ABB RAPID module: P51.mod

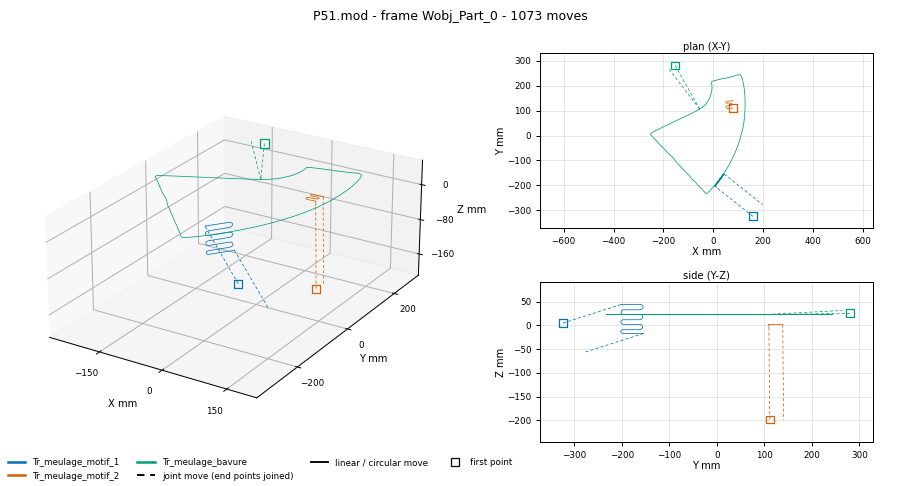
[picture p0: tool path of P51.mod in frame Wobj_Part_0, 1073 of 1081 moves have a stored position in this frame; points joined in program order, loops and branches not executed]
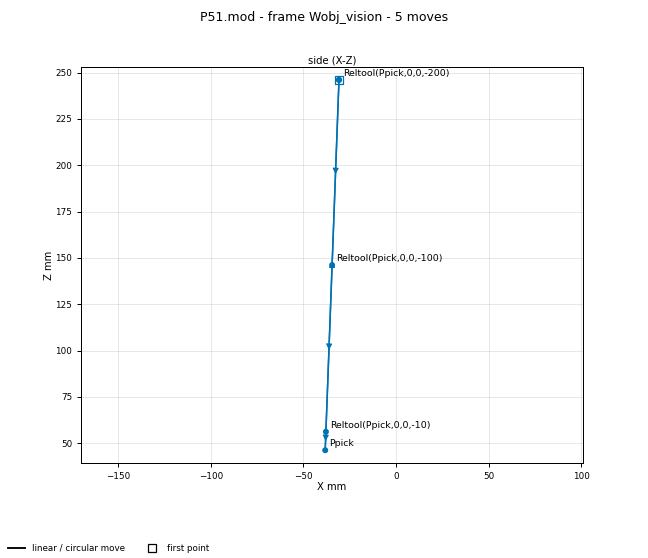
[picture p1: tool path of P51.mod in frame Wobj_vision, 5 of 1081 moves have a stored position in this frame; points joined in program order, loops and branches not executed]
MODULE P51
	LOCAL CONST Speeddata vitesse_Tronconnage :=[10, 500, 0, 0];
	LOCAL CONST Robtarget Tr_meulage_motif_1_App1 :=[[158.377655595794,-324.024414771468,4.86982949443898],[0.696320279376617,-0.571579290814731,-0.275420255163045,0.335527742350052],[0,0,0,0],[8.999999E+09,8.999999E+09,8.999999E+09,8.999999E+09,8.999999E+09,8.999999E+09]];
	LOCAL CONST Robtarget Tr_meulage_motif_1_App2 :=[[12.6243167397507,-207.899791051073,41.8973324903469],[0.696320279376617,-0.571579290814731,-0.275420255163045,0.335527742350052],[0,0,0,0],[8.999999E+09,8.999999E+09,8.999999E+09,8.999999E+09,8.999999E+09,8.999999E+09]];
	LOCAL CONST Robtarget Tr_meulage_motif_1_P0 :=[[4.95308837890625,-201.78796875,43.8461484375],[0.696320279376617,-0.571579290814731,-0.275420255163045,0.335527742350052],[0,0,0,0],[8.999999E+09,8.999999E+09,8.999999E+09,8.999999E+09,8.999999E+09,8.999999E+09]];
	LOCAL CONST Robtarget Tr_meulage_motif_1_P1 :=[[5.54933837890625,-200.985171875,43.84616796875],[0.696320279376617,-0.571579290814731,-0.275420255163045,0.335527742350052],[0,0,0,0],[8.999999E+09,8.999999E+09,8.999999E+09,8.999999E+09,8.999999E+09,8.999999E+09]];
	LOCAL CONST Robtarget Tr_meulage_motif_1_P2 :=[[6.1455888671875,-200.182375,43.8461875],[0.696320279376617,-0.571579290814731,-0.275420255163045,0.335527742350052],[0,0,0,0],[8.999999E+09,8.999999E+09,8.999999E+09,8.999999E+09,8.999999E+09,8.999999E+09]];
	LOCAL CONST Robtarget Tr_meulage_motif_1_P3 :=[[6.74183935546875,-199.379578125,43.84620703125],[0.696320279376617,-0.571579290814731,-0.275420255163045,0.335527742350052],[0,0,0,0],[8.999999E+09,8.999999E+09,8.999999E+09,8.999999E+09,8.999999E+09,8.999999E+09]];
	LOCAL CONST Robtarget Tr_meulage_motif_1_P4 :=[[7.33808935546875,-198.57678125,43.84623046875],[0.696320279376617,-0.571579290814731,-0.275420255163045,0.335527742350052],[0,0,0,0],[8.999999E+09,8.999999E+09,8.999999E+09,8.999999E+09,8.999999E+09,8.999999E+09]];
	LOCAL CONST Robtarget Tr_meulage_motif_1_P5 :=[[7.93433984375,-197.773984375,43.84625],[0.696320279376617,-0.571579290814731,-0.275420255163045,0.335527742350052],[0,0,0,0],[8.999999E+09,8.999999E+09,8.999999E+09,8.999999E+09,8.999999E+09,8.999999E+09]];
	LOCAL CONST Robtarget Tr_meulage_motif_1_P6 :=[[8.53058984375,-196.9711875,43.84626953125],[0.696320279376617,-0.571579290814731,-0.275420255163045,0.335527742350052],[0,0,0,0],[8.999999E+09,8.999999E+09,8.999999E+09,8.999999E+09,8.999999E+09,8.999999E+09]];
	LOCAL CONST Robtarget Tr_meulage_motif_1_P7 :=[[9.12683984375,-196.168390625,43.8462890625],[0.696320279376617,-0.571579290814731,-0.275420255163045,0.335527742350052],[0,0,0,0],[8.999999E+09,8.999999E+09,8.999999E+09,8.999999E+09,8.999999E+09,8.999999E+09]];
	LOCAL CONST Robtarget Tr_meulage_motif_1_P8 :=[[9.7230908203125,-195.36559375,43.84630859375],[0.696320279376617,-0.571579290814731,-0.275420255163045,0.335527742350052],[0,0,0,0],[8.999999E+09,8.999999E+09,8.999999E+09,8.999999E+09,8.999999E+09,8.999999E+09]];
	LOCAL CONST Robtarget Tr_meulage_motif_1_P9 :=[[10.3193408203125,-194.56278125,43.846328125],[0.696320279376617,-0.571579290814731,-0.275420255163045,0.335527742350052],[0,0,0,0],[8.999999E+09,8.999999E+09,8.999999E+09,8.999999E+09,8.999999E+09,8.999999E+09]];
	LOCAL CONST Robtarget Tr_meulage_motif_1_P10 :=[[10.9155908203125,-193.759984375,43.8463515625],[0.696320279376617,-0.571579290814731,-0.275420255163045,0.335527742350052],[0,0,0,0],[8.999999E+09,8.999999E+09,8.999999E+09,8.999999E+09,8.999999E+09,8.999999E+09]];
	LOCAL CONST Robtarget Tr_meulage_motif_1_P11 :=[[11.511841796875,-192.9571875,43.84637109375],[0.696320279376617,-0.571579290814731,-0.275420255163045,0.335527742350052],[0,0,0,0],[8.999999E+09,8.999999E+09,8.999999E+09,8.999999E+09,8.999999E+09,8.999999E+09]];
	LOCAL CONST Robtarget Tr_meulage_motif_1_P12 :=[[12.108091796875,-192.154390625,43.846390625],[0.696320279376617,-0.571579290814731,-0.275420255163045,0.335527742350052],[0,0,0,0],[8.999999E+09,8.999999E+09,8.999999E+09,8.999999E+09,8.999999E+09,8.999999E+09]];
	LOCAL CONST Robtarget Tr_meulage_motif_1_P13 :=[[12.704341796875,-191.35159375,43.84641015625],[0.696320279376617,-0.571579290814731,-0.275420255163045,0.335527742350052],[0,0,0,0],[8.999999E+09,8.999999E+09,8.999999E+09,8.999999E+09,8.999999E+09,8.999999E+09]];
	LOCAL CONST Robtarget Tr_meulage_motif_1_P14 :=[[13.3005927734375,-190.548796875,43.8464296875],[0.696320279376617,-0.571579290814731,-0.275420255163045,0.335527742350052],[0,0,0,0],[8.999999E+09,8.999999E+09,8.999999E+09,8.999999E+09,8.999999E+09,8.999999E+09]];
	LOCAL CONST Robtarget Tr_meulage_motif_1_P15 :=[[13.8968427734375,-189.746,43.846453125],[0.696320279376617,-0.571579290814731,-0.275420255163045,0.335527742350052],[0,0,0,0],[8.999999E+09,8.999999E+09,8.999999E+09,8.999999E+09,8.999999E+09,8.999999E+09]];
	LOCAL CONST Robtarget Tr_meulage_motif_1_P16 :=[[14.4930927734375,-188.943203125,43.84647265625],[0.696320279376617,-0.571579290814731,-0.275420255163045,0.335527742350052],[0,0,0,0],[8.999999E+09,8.999999E+09,8.999999E+09,8.999999E+09,8.999999E+09,8.999999E+09]];
	LOCAL CONST Robtarget Tr_meulage_motif_1_P17 :=[[15.0893427734375,-188.14040625,43.8464921875],[0.696320279376617,-0.571579290814731,-0.275420255163045,0.335527742350052],[0,0,0,0],[8.999999E+09,8.999999E+09,8.999999E+09,8.999999E+09,8.999999E+09,8.999999E+09]];
	LOCAL CONST Robtarget Tr_meulage_motif_1_P18 :=[[15.68559375,-187.33759375,43.84651171875],[0.696320279376617,-0.571579290814731,-0.275420255163045,0.335527742350052],[0,0,0,0],[8.999999E+09,8.999999E+09,8.999999E+09,8.999999E+09,8.999999E+09,8.999999E+09]];
	LOCAL CONST Robtarget Tr_meulage_motif_1_P19 :=[[16.28184375,-186.534796875,43.84653125],[0.696320279376617,-0.571579290814731,-0.275420255163045,0.335527742350052],[0,0,0,0],[8.999999E+09,8.999999E+09,8.999999E+09,8.999999E+09,8.999999E+09,8.999999E+09]];
	LOCAL CONST Robtarget Tr_meulage_motif_1_P20 :=[[16.87809375,-185.732,43.8465546875],[0.696320279376617,-0.571579290814731,-0.275420255163045,0.335527742350052],[0,0,0,0],[8.999999E+09,8.999999E+09,8.999999E+09,8.999999E+09,8.999999E+09,8.999999E+09]];
	LOCAL CONST Robtarget Tr_meulage_motif_1_P21 :=[[17.47434375,-184.929203125,43.84657421875],[0.696320279376617,-0.571579290814731,-0.275420255163045,0.335527742350052],[0,0,0,0],[8.999999E+09,8.999999E+09,8.999999E+09,8.999999E+09,8.999999E+09,8.999999E+09]];
	LOCAL CONST Robtarget Tr_meulage_motif_1_P22 :=[[18.07059375,-184.12640625,43.84659375],[0.696320279376617,-0.571579290814731,-0.275420255163045,0.335527742350052],[0,0,0,0],[8.999999E+09,8.999999E+09,8.999999E+09,8.999999E+09,8.999999E+09,8.999999E+09]];
	LOCAL CONST Robtarget Tr_meulage_motif_1_P23 :=[[18.666845703125,-183.323609375,43.84661328125],[0.696320279376617,-0.571579290814731,-0.275420255163045,0.335527742350052],[0,0,0,0],[8.999999E+09,8.999999E+09,8.999999E+09,8.999999E+09,8.999999E+09,8.999999E+09]];
	LOCAL CONST Robtarget Tr_meulage_motif_1_P24 :=[[19.263095703125,-182.5208125,43.8466328125],[0.696320279376617,-0.571579290814731,-0.275420255163045,0.335527742350052],[0,0,0,0],[8.999999E+09,8.999999E+09,8.999999E+09,8.999999E+09,8.999999E+09,8.999999E+09]];
	LOCAL CONST Robtarget Tr_meulage_motif_1_P25 :=[[19.859345703125,-181.718015625,43.84665234375],[0.696320279376617,-0.571579290814731,-0.275420255163045,0.335527742350052],[0,0,0,0],[8.999999E+09,8.999999E+09,8.999999E+09,8.999999E+09,8.999999E+09,8.999999E+09]];
	LOCAL CONST Robtarget Tr_meulage_motif_1_P26 :=[[20.455595703125,-180.91521875,43.84667578125],[0.696320279376617,-0.571579290814731,-0.275420255163045,0.335527742350052],[0,0,0,0],[8.999999E+09,8.999999E+09,8.999999E+09,8.999999E+09,8.999999E+09,8.999999E+09]];
	LOCAL CONST Robtarget Tr_meulage_motif_1_P27 :=[[21.051845703125,-180.11240625,43.8466953125],[0.696320279376617,-0.571579290814731,-0.275420255163045,0.335527742350052],[0,0,0,0],[8.999999E+09,8.999999E+09,8.999999E+09,8.999999E+09,8.999999E+09,8.999999E+09]];
	LOCAL CONST Robtarget Tr_meulage_motif_1_P28 :=[[21.648095703125,-179.309609375,43.84671484375],[0.696320279376617,-0.571579290814731,-0.275420255163045,0.335527742350052],[0,0,0,0],[8.999999E+09,8.999999E+09,8.999999E+09,8.999999E+09,8.999999E+09,8.999999E+09]];
	LOCAL CONST Robtarget Tr_meulage_motif_1_P29 :=[[22.24434765625,-178.5068125,43.846734375],[0.696320279376617,-0.571579290814731,-0.275420255163045,0.335527742350052],[0,0,0,0],[8.999999E+09,8.999999E+09,8.999999E+09,8.999999E+09,8.999999E+09,8.999999E+09]];
	LOCAL CONST Robtarget Tr_meulage_motif_1_P30 :=[[22.84059765625,-177.704015625,43.84675390625],[0.696320279376617,-0.571579290814731,-0.275420255163045,0.335527742350052],[0,0,0,0],[8.999999E+09,8.999999E+09,8.999999E+09,8.999999E+09,8.999999E+09,8.999999E+09]];
	LOCAL CONST Robtarget Tr_meulage_motif_1_P31 :=[[23.43684765625,-176.90121875,43.84677734375],[0.696320279376617,-0.571579290814731,-0.275420255163045,0.335527742350052],[0,0,0,0],[8.999999E+09,8.999999E+09,8.999999E+09,8.999999E+09,8.999999E+09,8.999999E+09]];
	LOCAL CONST Robtarget Tr_meulage_motif_1_P32 :=[[24.03309765625,-176.098421875,43.846796875],[0.696320279376617,-0.571579290814731,-0.275420255163045,0.335527742350052],[0,0,0,0],[8.999999E+09,8.999999E+09,8.999999E+09,8.999999E+09,8.999999E+09,8.999999E+09]];
	LOCAL CONST Robtarget Tr_meulage_motif_1_P33 :=[[24.62934765625,-175.295625,43.84681640625],[0.696320279376617,-0.571579290814731,-0.275420255163045,0.335527742350052],[0,0,0,0],[8.999999E+09,8.999999E+09,8.999999E+09,8.999999E+09,8.999999E+09,8.999999E+09]];
	LOCAL CONST Robtarget Tr_meulage_motif_1_P34 :=[[25.22559765625,-174.492828125,43.8468359375],[0.696320279376617,-0.571579290814731,-0.275420255163045,0.335527742350052],[0,0,0,0],[8.999999E+09,8.999999E+09,8.999999E+09,8.999999E+09,8.999999E+09,8.999999E+09]];
	LOCAL CONST Robtarget Tr_meulage_motif_1_P35 :=[[25.82184765625,-173.69003125,43.84685546875],[0.696320279376617,-0.571579290814731,-0.275420255163045,0.335527742350052],[0,0,0,0],[8.999999E+09,8.999999E+09,8.999999E+09,8.999999E+09,8.999999E+09,8.999999E+09]];
	LOCAL CONST Robtarget Tr_meulage_motif_1_P36 :=[[26.418099609375,-172.887234375,43.84687890625],[0.696320279376617,-0.571579290814731,-0.275420255163045,0.335527742350052],[0,0,0,0],[8.999999E+09,8.999999E+09,8.999999E+09,8.999999E+09,8.999999E+09,8.999999E+09]];
	LOCAL CONST Robtarget Tr_meulage_motif_1_P37 :=[[27.014349609375,-172.084421875,43.8468984375],[0.696320279376617,-0.571579290814731,-0.275420255163045,0.335527742350052],[0,0,0,0],[8.999999E+09,8.999999E+09,8.999999E+09,8.999999E+09,8.999999E+09,8.999999E+09]];
	LOCAL CONST Robtarget Tr_meulage_motif_1_P38 :=[[27.610599609375,-171.281625,43.84691796875],[0.696320279376617,-0.571579290814731,-0.275420255163045,0.335527742350052],[0,0,0,0],[8.999999E+09,8.999999E+09,8.999999E+09,8.999999E+09,8.999999E+09,8.999999E+09]];
	LOCAL CONST Robtarget Tr_meulage_motif_1_P39 :=[[28.206849609375,-170.478828125,43.8469375],[0.696320279376617,-0.571579290814731,-0.275420255163045,0.335527742350052],[0,0,0,0],[8.999999E+09,8.999999E+09,8.999999E+09,8.999999E+09,8.999999E+09,8.999999E+09]];
	LOCAL CONST Robtarget Tr_meulage_motif_1_P40 :=[[28.803099609375,-169.67603125,43.84695703125],[0.696320279376617,-0.571579290814731,-0.275420255163045,0.335527742350052],[0,0,0,0],[8.999999E+09,8.999999E+09,8.999999E+09,8.999999E+09,8.999999E+09,8.999999E+09]];
	LOCAL CONST Robtarget Tr_meulage_motif_1_P41 :=[[29.399349609375,-168.873234375,43.8469765625],[0.696320279376617,-0.571579290814731,-0.275420255163045,0.335527742350052],[0,0,0,0],[8.999999E+09,8.999999E+09,8.999999E+09,8.999999E+09,8.999999E+09,8.999999E+09]];
	LOCAL CONST Robtarget Tr_meulage_motif_1_P42 :=[[29.995599609375,-168.0704375,43.847],[0.696320279376617,-0.571579290814731,-0.275420255163045,0.335527742350052],[0,0,0,0],[8.999999E+09,8.999999E+09,8.999999E+09,8.999999E+09,8.999999E+09,8.999999E+09]];
	LOCAL CONST Robtarget Tr_meulage_motif_1_P43 :=[[30.5918515625,-167.267640625,43.84701953125],[0.696320279376617,-0.571579290814731,-0.275420255163045,0.335527742350052],[0,0,0,0],[8.999999E+09,8.999999E+09,8.999999E+09,8.999999E+09,8.999999E+09,8.999999E+09]];
	LOCAL CONST Robtarget Tr_meulage_motif_1_P44 :=[[31.1881015625,-166.46484375,43.8470390625],[0.696320279376617,-0.571579290814731,-0.275420255163045,0.335527742350052],[0,0,0,0],[8.999999E+09,8.999999E+09,8.999999E+09,8.999999E+09,8.999999E+09,8.999999E+09]];
	LOCAL CONST Robtarget Tr_meulage_motif_1_P45 :=[[31.7843515625,-165.662046875,43.84705859375],[0.696320279376617,-0.571579290814731,-0.275420255163045,0.335527742350052],[0,0,0,0],[8.999999E+09,8.999999E+09,8.999999E+09,8.999999E+09,8.999999E+09,8.999999E+09]];
	LOCAL CONST Robtarget Tr_meulage_motif_1_P46 :=[[32.3806015625,-164.859234375,43.847078125],[0.696320279376617,-0.571579290814731,-0.275420255163045,0.335527742350052],[0,0,0,0],[8.999999E+09,8.999999E+09,8.999999E+09,8.999999E+09,8.999999E+09,8.999999E+09]];
	LOCAL CONST Robtarget Tr_meulage_motif_1_P47 :=[[32.9768515625,-164.0564375,43.8471015625],[0.696320279376617,-0.571579290814731,-0.275420255163045,0.335527742350052],[0,0,0,0],[8.999999E+09,8.999999E+09,8.999999E+09,8.999999E+09,8.999999E+09,8.999999E+09]];
	LOCAL CONST Robtarget Tr_meulage_motif_1_P48 :=[[33.5731015625,-163.253640625,43.84712109375],[0.696320279376617,-0.571579290814731,-0.275420255163045,0.335527742350052],[0,0,0,0],[8.999999E+09,8.999999E+09,8.999999E+09,8.999999E+09,8.999999E+09,8.999999E+09]];
	LOCAL CONST Robtarget Tr_meulage_motif_1_P49 :=[[34.1693515625,-162.45084375,43.847140625],[0.696320279376617,-0.571579290814731,-0.275420255163045,0.335527742350052],[0,0,0,0],[8.999999E+09,8.999999E+09,8.999999E+09,8.999999E+09,8.999999E+09,8.999999E+09]];
	LOCAL CONST Robtarget Tr_meulage_motif_1_P50 :=[[34.7656015625,-161.648046875,43.84716015625],[0.696320279376617,-0.571579290814731,-0.275420255163045,0.335527742350052],[0,0,0,0],[8.999999E+09,8.999999E+09,8.999999E+09,8.999999E+09,8.999999E+09,8.999999E+09]];
	LOCAL CONST Robtarget Tr_meulage_motif_1_P51 :=[[35.3618515625,-160.84525,43.8471796875],[0.696320279376617,-0.571579290814731,-0.275420255163045,0.335527742350052],[0,0,0,0],[8.999999E+09,8.999999E+09,8.999999E+09,8.999999E+09,8.999999E+09,8.999999E+09]];
	LOCAL CONST Robtarget Tr_meulage_motif_1_P52 :=[[35.957796875,-160.051484375,43.7367265625],[0.696320279376617,-0.571579290814731,-0.275420255163045,0.335527742350052],[0,0,0,0],[8.999999E+09,8.999999E+09,8.999999E+09,8.999999E+09,8.999999E+09,8.999999E+09]];
	LOCAL CONST Robtarget Tr_meulage_motif_1_P53 :=[[36.53003125,-159.297484375,43.52578515625],[0.696320279376617,-0.571579290814731,-0.275420255163045,0.335527742350052],[0,0,0,0],[8.999999E+09,8.999999E+09,8.999999E+09,8.999999E+09,8.999999E+09,8.999999E+09]];
	LOCAL CONST Robtarget Tr_meulage_motif_1_P54 :=[[37.04861328125,-158.620453125,43.25425390625],[0.696320279376617,-0.571579290814731,-0.275420255163045,0.335527742350052],[0,0,0,0],[8.999999E+09,8.999999E+09,8.999999E+09,8.999999E+09,8.999999E+09,8.999999E+09]];
	LOCAL CONST Robtarget Tr_meulage_motif_1_P55 :=[[37.5060625,-158.026046875,42.97862890625],[0.696320279376617,-0.571579290814731,-0.275420255163045,0.335527742350052],[0,0,0,0],[8.999999E+09,8.999999E+09,8.999999E+09,8.999999E+09,8.999999E+09,8.999999E+09]];
	LOCAL CONST Robtarget Tr_meulage_motif_1_P56 :=[[38.1855703125,-157.1591875,42.36319140625],[0.696320279376617,-0.571579290814731,-0.275420255163045,0.335527742350052],[0,0,0,0],[8.999999E+09,8.999999E+09,8.999999E+09,8.999999E+09,8.999999E+09,8.999999E+09]];
	LOCAL CONST Robtarget Tr_meulage_motif_1_P57 :=[[38.8276953125,-156.3606875,41.51647265625],[0.696320279376617,-0.571579290814731,-0.275420255163045,0.335527742350052],[0,0,0,0],[8.999999E+09,8.999999E+09,8.999999E+09,8.999999E+09,8.999999E+09,8.999999E+09]];
	LOCAL CONST Robtarget Tr_meulage_motif_1_P58 :=[[39.371328125,-155.7085625,40.49372265625],[0.696320279376617,-0.571579290814731,-0.275420255163045,0.335527742350052],[0,0,0,0],[8.999999E+09,8.999999E+09,8.999999E+09,8.999999E+09,8.999999E+09,8.999999E+09]];
	LOCAL CONST Robtarget Tr_meulage_motif_1_P59 :=[[39.7040546875,-155.347578125,39.37875],[0.696320279376617,-0.571579290814731,-0.275420255163045,0.335527742350052],[0,0,0,0],[8.999999E+09,8.999999E+09,8.999999E+09,8.999999E+09,8.999999E+09,8.999999E+09]];
	LOCAL CONST Robtarget Tr_meulage_motif_1_P60 :=[[39.74616796875,-155.345125,38.68353515625],[0.696320279376617,-0.571579290814731,-0.275420255163045,0.335527742350052],[0,0,0,0],[8.999999E+09,8.999999E+09,8.999999E+09,8.999999E+09,8.999999E+09,8.999999E+09]];
	LOCAL CONST Robtarget Tr_meulage_motif_1_P61 :=[[39.7708515625,-155.363453125,38.023],[0.696320279376617,-0.571579290814731,-0.275420255163045,0.335527742350052],[0,0,0,0],[8.999999E+09,8.999999E+09,8.999999E+09,8.999999E+09,8.999999E+09,8.999999E+09]];
	LOCAL CONST Robtarget Tr_meulage_motif_1_P62 :=[[39.76280859375,-155.4258125,37.36262109375],[0.696320279376617,-0.571579290814731,-0.275420255163045,0.335527742350052],[0,0,0,0],[8.999999E+09,8.999999E+09,8.999999E+09,8.999999E+09,8.999999E+09,8.999999E+09]];
	LOCAL CONST Robtarget Tr_meulage_motif_1_P63 :=[[39.50687109375,-155.856296875,36.26205078125],[0.696320279376617,-0.571579290814731,-0.275420255163045,0.335527742350052],[0,0,0,0],[8.999999E+09,8.999999E+09,8.999999E+09,8.999999E+09,8.999999E+09,8.999999E+09]];
	LOCAL CONST Robtarget Tr_meulage_motif_1_P64 :=[[39.03368359375,-156.571875,35.25649609375],[0.696320279376617,-0.571579290814731,-0.275420255163045,0.335527742350052],[0,0,0,0],[8.999999E+09,8.999999E+09,8.999999E+09,8.999999E+09,8.999999E+09,8.999999E+09]];
	LOCAL CONST Robtarget Tr_meulage_motif_1_P65 :=[[38.4544140625,-157.416421875,34.42849609375],[0.696320279376617,-0.571579290814731,-0.275420255163045,0.335527742350052],[0,0,0,0],[8.999999E+09,8.999999E+09,8.999999E+09,8.999999E+09,8.999999E+09,8.999999E+09]];
	LOCAL CONST Robtarget Tr_meulage_motif_1_P66 :=[[38.0595078125,-157.978984375,34.03316015625],[0.696320279376617,-0.571579290814731,-0.275420255163045,0.335527742350052],[0,0,0,0],[8.999999E+09,8.999999E+09,8.999999E+09,8.999999E+09,8.999999E+09,8.999999E+09]];
	LOCAL CONST Robtarget Tr_meulage_motif_1_P67 :=[[37.38715234375,-158.92225,33.5461328125],[0.696320279376617,-0.571579290814731,-0.275420255163045,0.335527742350052],[0,0,0,0],[8.999999E+09,8.999999E+09,8.999999E+09,8.999999E+09,8.999999E+09,8.999999E+09]];
	LOCAL CONST Robtarget Tr_meulage_motif_1_P68 :=[[36.89316015625,-159.607953125,33.28230859375],[0.696320279376617,-0.571579290814731,-0.275420255163045,0.335527742350052],[0,0,0,0],[8.999999E+09,8.999999E+09,8.999999E+09,8.999999E+09,8.999999E+09,8.999999E+09]];
	LOCAL CONST Robtarget Tr_meulage_motif_1_P69 :=[[36.34508984375,-160.361828125,33.0780390625],[0.696320279376617,-0.571579290814731,-0.275420255163045,0.335527742350052],[0,0,0,0],[8.999999E+09,8.999999E+09,8.999999E+09,8.999999E+09,8.999999E+09,8.999999E+09]];
	LOCAL CONST Robtarget Tr_meulage_motif_1_P70 :=[[35.76388671875,-161.152828125,32.96954296875],[0.696320279376617,-0.571579290814731,-0.275420255163045,0.335527742350052],[0,0,0,0],[8.999999E+09,8.999999E+09,8.999999E+09,8.999999E+09,8.999999E+09,8.999999E+09]];
	LOCAL CONST Robtarget Tr_meulage_motif_1_P71 :=[[35.17619921875,-161.95271875,32.85905078125],[0.696320279376617,-0.571579290814731,-0.275420255163045,0.335527742350052],[0,0,0,0],[8.999999E+09,8.999999E+09,8.999999E+09,8.999999E+09,8.999999E+09,8.999999E+09]];
	LOCAL CONST Robtarget Tr_meulage_motif_1_P72 :=[[34.57994921875,-162.755515625,32.85903125],[0.696320279376617,-0.571579290814731,-0.275420255163045,0.335527742350052],[0,0,0,0],[8.999999E+09,8.999999E+09,8.999999E+09,8.999999E+09,8.999999E+09,8.999999E+09]];
	LOCAL CONST Robtarget Tr_meulage_motif_1_P73 :=[[33.9836953125,-163.558328125,32.8590078125],[0.696320279376617,-0.571579290814731,-0.275420255163045,0.335527742350052],[0,0,0,0],[8.999999E+09,8.999999E+09,8.999999E+09,8.999999E+09,8.999999E+09,8.999999E+09]];
	LOCAL CONST Robtarget Tr_meulage_motif_1_P74 :=[[33.3874453125,-164.361125,32.85898828125],[0.696320279376617,-0.571579290814731,-0.275420255163045,0.335527742350052],[0,0,0,0],[8.999999E+09,8.999999E+09,8.999999E+09,8.999999E+09,8.999999E+09,8.999999E+09]];
	LOCAL CONST Robtarget Tr_meulage_motif_1_P75 :=[[32.7911953125,-165.163921875,32.85896875],[0.696320279376617,-0.571579290814731,-0.275420255163045,0.335527742350052],[0,0,0,0],[8.999999E+09,8.999999E+09,8.999999E+09,8.999999E+09,8.999999E+09,8.999999E+09]];
	LOCAL CONST Robtarget Tr_meulage_motif_1_P76 :=[[32.1949453125,-165.96671875,32.85894921875],[0.696320279376617,-0.571579290814731,-0.275420255163045,0.335527742350052],[0,0,0,0],[8.999999E+09,8.999999E+09,8.999999E+09,8.999999E+09,8.999999E+09,8.999999E+09]];
	LOCAL CONST Robtarget Tr_meulage_motif_1_P77 :=[[31.5986953125,-166.769515625,32.8589296875],[0.696320279376617,-0.571579290814731,-0.275420255163045,0.335527742350052],[0,0,0,0],[8.999999E+09,8.999999E+09,8.999999E+09,8.999999E+09,8.999999E+09,8.999999E+09]];
	LOCAL CONST Robtarget Tr_meulage_motif_1_P78 :=[[31.0024453125,-167.5723125,32.85890625],[0.696320279376617,-0.571579290814731,-0.275420255163045,0.335527742350052],[0,0,0,0],[8.999999E+09,8.999999E+09,8.999999E+09,8.999999E+09,8.999999E+09,8.999999E+09]];
	LOCAL CONST Robtarget Tr_meulage_motif_1_P79 :=[[30.4061953125,-168.375109375,32.85888671875],[0.696320279376617,-0.571579290814731,-0.275420255163045,0.335527742350052],[0,0,0,0],[8.999999E+09,8.999999E+09,8.999999E+09,8.999999E+09,8.999999E+09,8.999999E+09]];
	LOCAL CONST Robtarget Tr_meulage_motif_1_P80 :=[[29.8099453125,-169.17790625,32.8588671875],[0.696320279376617,-0.571579290814731,-0.275420255163045,0.335527742350052],[0,0,0,0],[8.999999E+09,8.999999E+09,8.999999E+09,8.999999E+09,8.999999E+09,8.999999E+09]];
	LOCAL CONST Robtarget Tr_meulage_motif_1_P81 :=[[29.2136953125,-169.980703125,32.85884765625],[0.696320279376617,-0.571579290814731,-0.275420255163045,0.335527742350052],[0,0,0,0],[8.999999E+09,8.999999E+09,8.999999E+09,8.999999E+09,8.999999E+09,8.999999E+09]];
	LOCAL CONST Robtarget Tr_meulage_motif_1_P82 :=[[28.6174453125,-170.783515625,32.858828125],[0.696320279376617,-0.571579290814731,-0.275420255163045,0.335527742350052],[0,0,0,0],[8.999999E+09,8.999999E+09,8.999999E+09,8.999999E+09,8.999999E+09,8.999999E+09]];
	LOCAL CONST Robtarget Tr_meulage_motif_1_P83 :=[[28.021193359375,-171.5863125,32.8588046875],[0.696320279376617,-0.571579290814731,-0.275420255163045,0.335527742350052],[0,0,0,0],[8.999999E+09,8.999999E+09,8.999999E+09,8.999999E+09,8.999999E+09,8.999999E+09]];
	LOCAL CONST Robtarget Tr_meulage_motif_1_P84 :=[[27.424943359375,-172.389109375,32.85878515625],[0.696320279376617,-0.571579290814731,-0.275420255163045,0.335527742350052],[0,0,0,0],[8.999999E+09,8.999999E+09,8.999999E+09,8.999999E+09,8.999999E+09,8.999999E+09]];
	LOCAL CONST Robtarget Tr_meulage_motif_1_P85 :=[[26.828693359375,-173.19190625,32.858765625],[0.696320279376617,-0.571579290814731,-0.275420255163045,0.335527742350052],[0,0,0,0],[8.999999E+09,8.999999E+09,8.999999E+09,8.999999E+09,8.999999E+09,8.999999E+09]];
	LOCAL CONST Robtarget Tr_meulage_motif_1_P86 :=[[26.232443359375,-173.994703125,32.85874609375],[0.696320279376617,-0.571579290814731,-0.275420255163045,0.335527742350052],[0,0,0,0],[8.999999E+09,8.999999E+09,8.999999E+09,8.999999E+09,8.999999E+09,8.999999E+09]];
	LOCAL CONST Robtarget Tr_meulage_motif_1_P87 :=[[25.636193359375,-174.7975,32.8587265625],[0.696320279376617,-0.571579290814731,-0.275420255163045,0.335527742350052],[0,0,0,0],[8.999999E+09,8.999999E+09,8.999999E+09,8.999999E+09,8.999999E+09,8.999999E+09]];
	LOCAL CONST Robtarget Tr_meulage_motif_1_P88 :=[[25.039943359375,-175.600296875,32.85870703125],[0.696320279376617,-0.571579290814731,-0.275420255163045,0.335527742350052],[0,0,0,0],[8.999999E+09,8.999999E+09,8.999999E+09,8.999999E+09,8.999999E+09,8.999999E+09]];
	LOCAL CONST Robtarget Tr_meulage_motif_1_P89 :=[[24.44369140625,-176.40309375,32.85868359375],[0.696320279376617,-0.571579290814731,-0.275420255163045,0.335527742350052],[0,0,0,0],[8.999999E+09,8.999999E+09,8.999999E+09,8.999999E+09,8.999999E+09,8.999999E+09]];
	LOCAL CONST Robtarget Tr_meulage_motif_1_P90 :=[[23.84744140625,-177.205890625,32.8586640625],[0.696320279376617,-0.571579290814731,-0.275420255163045,0.335527742350052],[0,0,0,0],[8.999999E+09,8.999999E+09,8.999999E+09,8.999999E+09,8.999999E+09,8.999999E+09]];
	LOCAL CONST Robtarget Tr_meulage_motif_1_P91 :=[[23.25119140625,-178.008703125,32.85864453125],[0.696320279376617,-0.571579290814731,-0.275420255163045,0.335527742350052],[0,0,0,0],[8.999999E+09,8.999999E+09,8.999999E+09,8.999999E+09,8.999999E+09,8.999999E+09]];
	LOCAL CONST Robtarget Tr_meulage_motif_1_P92 :=[[22.65494140625,-178.8115,32.858625],[0.696320279376617,-0.571579290814731,-0.275420255163045,0.335527742350052],[0,0,0,0],[8.999999E+09,8.999999E+09,8.999999E+09,8.999999E+09,8.999999E+09,8.999999E+09]];
	LOCAL CONST Robtarget Tr_meulage_motif_1_P93 :=[[22.05869140625,-179.614296875,32.85860546875],[0.696320279376617,-0.571579290814731,-0.275420255163045,0.335527742350052],[0,0,0,0],[8.999999E+09,8.999999E+09,8.999999E+09,8.999999E+09,8.999999E+09,8.999999E+09]];
	LOCAL CONST Robtarget Tr_meulage_motif_1_P94 :=[[21.46244140625,-180.41709375,32.85858203125],[0.696320279376617,-0.571579290814731,-0.275420255163045,0.335527742350052],[0,0,0,0],[8.999999E+09,8.999999E+09,8.999999E+09,8.999999E+09,8.999999E+09,8.999999E+09]];
	LOCAL CONST Robtarget Tr_meulage_motif_1_P95 :=[[20.86619140625,-181.219890625,32.8585625],[0.696320279376617,-0.571579290814731,-0.275420255163045,0.335527742350052],[0,0,0,0],[8.999999E+09,8.999999E+09,8.999999E+09,8.999999E+09,8.999999E+09,8.999999E+09]];
	LOCAL CONST Robtarget Tr_meulage_motif_1_P96 :=[[20.269939453125,-182.0226875,32.85854296875],[0.696320279376617,-0.571579290814731,-0.275420255163045,0.335527742350052],[0,0,0,0],[8.999999E+09,8.999999E+09,8.999999E+09,8.999999E+09,8.999999E+09,8.999999E+09]];
	LOCAL CONST Robtarget Tr_meulage_motif_1_P97 :=[[19.673689453125,-182.825484375,32.8585234375],[0.696320279376617,-0.571579290814731,-0.275420255163045,0.335527742350052],[0,0,0,0],[8.999999E+09,8.999999E+09,8.999999E+09,8.999999E+09,8.999999E+09,8.999999E+09]];
	LOCAL CONST Robtarget Tr_meulage_motif_1_P98 :=[[19.077439453125,-183.62828125,32.85850390625],[0.696320279376617,-0.571579290814731,-0.275420255163045,0.335527742350052],[0,0,0,0],[8.999999E+09,8.999999E+09,8.999999E+09,8.999999E+09,8.999999E+09,8.999999E+09]];
	LOCAL CONST Robtarget Tr_meulage_motif_1_P99 :=[[18.481189453125,-184.431078125,32.85848046875],[0.696320279376617,-0.571579290814731,-0.275420255163045,0.335527742350052],[0,0,0,0],[8.999999E+09,8.999999E+09,8.999999E+09,8.999999E+09,8.999999E+09,8.999999E+09]];
	LOCAL CONST Robtarget Tr_meulage_motif_1_P100 :=[[17.884939453125,-185.233890625,32.8584609375],[0.696320279376617,-0.571579290814731,-0.275420255163045,0.335527742350052],[0,0,0,0],[8.999999E+09,8.999999E+09,8.999999E+09,8.999999E+09,8.999999E+09,8.999999E+09]];
	LOCAL CONST Robtarget Tr_meulage_motif_1_P101 :=[[17.288689453125,-186.0366875,32.85844140625],[0.696320279376617,-0.571579290814731,-0.275420255163045,0.335527742350052],[0,0,0,0],[8.999999E+09,8.999999E+09,8.999999E+09,8.999999E+09,8.999999E+09,8.999999E+09]];
	LOCAL CONST Robtarget Tr_meulage_motif_1_P102 :=[[16.692439453125,-186.839484375,32.858421875],[0.696320279376617,-0.571579290814731,-0.275420255163045,0.335527742350052],[0,0,0,0],[8.999999E+09,8.999999E+09,8.999999E+09,8.999999E+09,8.999999E+09,8.999999E+09]];
	LOCAL CONST Robtarget Tr_meulage_motif_1_P103 :=[[16.0961884765625,-187.64228125,32.85840234375],[0.696320279376617,-0.571579290814731,-0.275420255163045,0.335527742350052],[0,0,0,0],[8.999999E+09,8.999999E+09,8.999999E+09,8.999999E+09,8.999999E+09,8.999999E+09]];
	LOCAL CONST Robtarget Tr_meulage_motif_1_P104 :=[[15.4999384765625,-188.445078125,32.8583828125],[0.696320279376617,-0.571579290814731,-0.275420255163045,0.335527742350052],[0,0,0,0],[8.999999E+09,8.999999E+09,8.999999E+09,8.999999E+09,8.999999E+09,8.999999E+09]];
	LOCAL CONST Robtarget Tr_meulage_motif_1_P105 :=[[14.9036875,-189.247875,32.858359375],[0.696320279376617,-0.571579290814731,-0.275420255163045,0.335527742350052],[0,0,0,0],[8.999999E+09,8.999999E+09,8.999999E+09,8.999999E+09,8.999999E+09,8.999999E+09]];
	LOCAL CONST Robtarget Tr_meulage_motif_1_P106 :=[[14.3074375,-190.050671875,32.85833984375],[0.696320279376617,-0.571579290814731,-0.275420255163045,0.335527742350052],[0,0,0,0],[8.999999E+09,8.999999E+09,8.999999E+09,8.999999E+09,8.999999E+09,8.999999E+09]];
	LOCAL CONST Robtarget Tr_meulage_motif_1_P107 :=[[13.7111875,-190.85346875,32.8583203125],[0.696320279376617,-0.571579290814731,-0.275420255163045,0.335527742350052],[0,0,0,0],[8.999999E+09,8.999999E+09,8.999999E+09,8.999999E+09,8.999999E+09,8.999999E+09]];
	LOCAL CONST Robtarget Tr_meulage_motif_1_P108 :=[[13.1149365234375,-191.656265625,32.85830078125],[0.696320279376617,-0.571579290814731,-0.275420255163045,0.335527742350052],[0,0,0,0],[8.999999E+09,8.999999E+09,8.999999E+09,8.999999E+09,8.999999E+09,8.999999E+09]];
	LOCAL CONST Robtarget Tr_meulage_motif_1_P109 :=[[12.5186865234375,-192.459078125,32.85828125],[0.696320279376617,-0.571579290814731,-0.275420255163045,0.335527742350052],[0,0,0,0],[8.999999E+09,8.999999E+09,8.999999E+09,8.999999E+09,8.999999E+09,8.999999E+09]];
	LOCAL CONST Robtarget Tr_meulage_motif_1_P110 :=[[11.9224365234375,-193.261875,32.8582578125],[0.696320279376617,-0.571579290814731,-0.275420255163045,0.335527742350052],[0,0,0,0],[8.999999E+09,8.999999E+09,8.999999E+09,8.999999E+09,8.999999E+09,8.999999E+09]];
	LOCAL CONST Robtarget Tr_meulage_motif_1_P111 :=[[11.326185546875,-194.064671875,32.85823828125],[0.696320279376617,-0.571579290814731,-0.275420255163045,0.335527742350052],[0,0,0,0],[8.999999E+09,8.999999E+09,8.999999E+09,8.999999E+09,8.999999E+09,8.999999E+09]];
	LOCAL CONST Robtarget Tr_meulage_motif_1_P112 :=[[10.729935546875,-194.86746875,32.85821875],[0.696320279376617,-0.571579290814731,-0.275420255163045,0.335527742350052],[0,0,0,0],[8.999999E+09,8.999999E+09,8.999999E+09,8.999999E+09,8.999999E+09,8.999999E+09]];
	LOCAL CONST Robtarget Tr_meulage_motif_1_P113 :=[[10.133685546875,-195.670265625,32.85819921875],[0.696320279376617,-0.571579290814731,-0.275420255163045,0.335527742350052],[0,0,0,0],[8.999999E+09,8.999999E+09,8.999999E+09,8.999999E+09,8.999999E+09,8.999999E+09]];
	LOCAL CONST Robtarget Tr_meulage_motif_1_P114 :=[[9.537435546875,-196.4730625,32.8581796875],[0.696320279376617,-0.571579290814731,-0.275420255163045,0.335527742350052],[0,0,0,0],[8.999999E+09,8.999999E+09,8.999999E+09,8.999999E+09,8.999999E+09,8.999999E+09]];
	LOCAL CONST Robtarget Tr_meulage_motif_1_P115 :=[[8.9497470703125,-197.272953125,32.74768359375],[0.696320279376617,-0.571579290814731,-0.275420255163045,0.335527742350052],[0,0,0,0],[8.999999E+09,8.999999E+09,8.999999E+09,8.999999E+09,8.999999E+09,8.999999E+09]];
	LOCAL CONST Robtarget Tr_meulage_motif_1_P116 :=[[8.393279296875,-198.03865625,32.536705078125],[0.696320279376617,-0.571579290814731,-0.275420255163045,0.335527742350052],[0,0,0,0],[8.999999E+09,8.999999E+09,8.999999E+09,8.999999E+09,8.999999E+09,8.999999E+09]];
	LOCAL CONST Robtarget Tr_meulage_motif_1_P117 :=[[7.89499267578125,-198.73075,32.265138671875],[0.696320279376617,-0.571579290814731,-0.275420255163045,0.335527742350052],[0,0,0,0],[8.999999E+09,8.999999E+09,8.999999E+09,8.999999E+09,8.999999E+09,8.999999E+09]];
	LOCAL CONST Robtarget Tr_meulage_motif_1_P118 :=[[7.48211376953125,-199.310359375,31.961296875],[0.696320279376617,-0.571579290814731,-0.275420255163045,0.335527742350052],[0,0,0,0],[8.999999E+09,8.999999E+09,8.999999E+09,8.999999E+09,8.999999E+09,8.999999E+09]];
	LOCAL CONST Robtarget Tr_meulage_motif_1_P119 :=[[6.8900419921875,-200.1591875,31.2994609375],[0.696320279376617,-0.571579290814731,-0.275420255163045,0.335527742350052],[0,0,0,0],[8.999999E+09,8.999999E+09,8.999999E+09,8.999999E+09,8.999999E+09,8.999999E+09]];
	LOCAL CONST Robtarget Tr_meulage_motif_1_P120 :=[[6.385927734375,-200.908234375,30.398478515625],[0.696320279376617,-0.571579290814731,-0.275420255163045,0.335527742350052],[0,0,0,0],[8.999999E+09,8.999999E+09,8.999999E+09,8.999999E+09,8.999999E+09,8.999999E+09]];
	LOCAL CONST Robtarget Tr_meulage_motif_1_P121 :=[[6.10599755859375,-201.3666875,29.353568359375],[0.696320279376617,-0.571579290814731,-0.275420255163045,0.335527742350052],[0,0,0,0],[8.999999E+09,8.999999E+09,8.999999E+09,8.999999E+09,8.999999E+09,8.999999E+09]];
	LOCAL CONST Robtarget Tr_meulage_motif_1_P122 :=[[6.021697265625,-201.53421875,28.66109375],[0.696320279376617,-0.571579290814731,-0.275420255163045,0.335527742350052],[0,0,0,0],[8.999999E+09,8.999999E+09,8.999999E+09,8.999999E+09,8.999999E+09,8.999999E+09]];
	LOCAL CONST Robtarget Tr_meulage_motif_1_P123 :=[[6.0123720703125,-201.6068125,27.89192578125],[0.696320279376617,-0.571579290814731,-0.275420255163045,0.335527742350052],[0,0,0,0],[8.999999E+09,8.999999E+09,8.999999E+09,8.999999E+09,8.999999E+09,8.999999E+09]];
	LOCAL CONST Robtarget Tr_meulage_motif_1_P124 :=[[6.0810205078125,-201.574390625,27.122884765625],[0.696320279376617,-0.571579290814731,-0.275420255163045,0.335527742350052],[0,0,0,0],[8.999999E+09,8.999999E+09,8.999999E+09,8.999999E+09,8.999999E+09,8.999999E+09]];
	LOCAL CONST Robtarget Tr_meulage_motif_1_P125 :=[[6.37257080078125,-201.268234375,26.01583984375],[0.696320279376617,-0.571579290814731,-0.275420255163045,0.335527742350052],[0,0,0,0],[8.999999E+09,8.999999E+09,8.999999E+09,8.999999E+09,8.999999E+09,8.999999E+09]];
	LOCAL CONST Robtarget Tr_meulage_motif_1_P126 :=[[6.641466796875,-200.951859375,25.430794921875],[0.696320279376617,-0.571579290814731,-0.275420255163045,0.335527742350052],[0,0,0,0],[8.999999E+09,8.999999E+09,8.999999E+09,8.999999E+09,8.999999E+09,8.999999E+09]];
	LOCAL CONST Robtarget Tr_meulage_motif_1_P127 :=[[7.20352880859375,-200.264234375,24.544646484375],[0.696320279376617,-0.571579290814731,-0.275420255163045,0.335527742350052],[0,0,0,0],[8.999999E+09,8.999999E+09,8.999999E+09,8.999999E+09,8.999999E+09,8.999999E+09]];
	LOCAL CONST Robtarget Tr_meulage_motif_1_P128 :=[[7.5682099609375,-199.80553125,24.13079296875],[0.696320279376617,-0.571579290814731,-0.275420255163045,0.335527742350052],[0,0,0,0],[8.999999E+09,8.999999E+09,8.999999E+09,8.999999E+09,8.999999E+09,8.999999E+09]];
	LOCAL CONST Robtarget Tr_meulage_motif_1_P129 :=[[8.2550712890625,-198.923140625,23.587310546875],[0.696320279376617,-0.571579290814731,-0.275420255163045,0.335527742350052],[0,0,0,0],[8.999999E+09,8.999999E+09,8.999999E+09,8.999999E+09,8.999999E+09,8.999999E+09]];
	LOCAL CONST Robtarget Tr_meulage_motif_1_P130 :=[[8.758361328125,-198.268546875,23.292146484375],[0.696320279376617,-0.571579290814731,-0.275420255163045,0.335527742350052],[0,0,0,0],[8.999999E+09,8.999999E+09,8.999999E+09,8.999999E+09,8.999999E+09,8.999999E+09]];
	LOCAL CONST Robtarget Tr_meulage_motif_1_P131 :=[[9.32169921875,-197.526,23.08791796875],[0.696320279376617,-0.571579290814731,-0.275420255163045,0.335527742350052],[0,0,0,0],[8.999999E+09,8.999999E+09,8.999999E+09,8.999999E+09,8.999999E+09,8.999999E+09]];
	LOCAL CONST Robtarget Tr_meulage_motif_1_P132 :=[[9.911009765625,-196.741015625,22.9794609375],[0.696320279376617,-0.571579290814731,-0.275420255163045,0.335527742350052],[0,0,0,0],[8.999999E+09,8.999999E+09,8.999999E+09,8.999999E+09,8.999999E+09,8.999999E+09]];
	LOCAL CONST Robtarget Tr_meulage_motif_1_P133 :=[[10.506953125,-195.94725,22.869005859375],[0.696320279376617,-0.571579290814731,-0.275420255163045,0.335527742350052],[0,0,0,0],[8.999999E+09,8.999999E+09,8.999999E+09,8.999999E+09,8.999999E+09,8.999999E+09]];
	LOCAL CONST Robtarget Tr_meulage_motif_1_P134 :=[[11.1032041015625,-195.144453125,22.86902734375],[0.696320279376617,-0.571579290814731,-0.275420255163045,0.335527742350052],[0,0,0,0],[8.999999E+09,8.999999E+09,8.999999E+09,8.999999E+09,8.999999E+09,8.999999E+09]];
	LOCAL CONST Robtarget Tr_meulage_motif_1_P135 :=[[11.6994541015625,-194.341640625,22.869046875],[0.696320279376617,-0.571579290814731,-0.275420255163045,0.335527742350052],[0,0,0,0],[8.999999E+09,8.999999E+09,8.999999E+09,8.999999E+09,8.999999E+09,8.999999E+09]];
	LOCAL CONST Robtarget Tr_meulage_motif_1_P136 :=[[12.2957041015625,-193.53884375,22.869068359375],[0.696320279376617,-0.571579290814731,-0.275420255163045,0.335527742350052],[0,0,0,0],[8.999999E+09,8.999999E+09,8.999999E+09,8.999999E+09,8.999999E+09,8.999999E+09]];
	LOCAL CONST Robtarget Tr_meulage_motif_1_P137 :=[[12.8919541015625,-192.736046875,22.869087890625],[0.696320279376617,-0.571579290814731,-0.275420255163045,0.335527742350052],[0,0,0,0],[8.999999E+09,8.999999E+09,8.999999E+09,8.999999E+09,8.999999E+09,8.999999E+09]];
	LOCAL CONST Robtarget Tr_meulage_motif_1_P138 :=[[13.488205078125,-191.93325,22.869107421875],[0.696320279376617,-0.571579290814731,-0.275420255163045,0.335527742350052],[0,0,0,0],[8.999999E+09,8.999999E+09,8.999999E+09,8.999999E+09,8.999999E+09,8.999999E+09]];
	LOCAL CONST Robtarget Tr_meulage_motif_1_P139 :=[[14.084455078125,-191.130453125,22.86912890625],[0.696320279376617,-0.571579290814731,-0.275420255163045,0.335527742350052],[0,0,0,0],[8.999999E+09,8.999999E+09,8.999999E+09,8.999999E+09,8.999999E+09,8.999999E+09]];
	LOCAL CONST Robtarget Tr_meulage_motif_1_P140 :=[[14.680705078125,-190.32765625,22.8691484375],[0.696320279376617,-0.571579290814731,-0.275420255163045,0.335527742350052],[0,0,0,0],[8.999999E+09,8.999999E+09,8.999999E+09,8.999999E+09,8.999999E+09,8.999999E+09]];
	LOCAL CONST Robtarget Tr_meulage_motif_1_P141 :=[[15.2769560546875,-189.524859375,22.86916796875],[0.696320279376617,-0.571579290814731,-0.275420255163045,0.335527742350052],[0,0,0,0],[8.999999E+09,8.999999E+09,8.999999E+09,8.999999E+09,8.999999E+09,8.999999E+09]];
	LOCAL CONST Robtarget Tr_meulage_motif_1_P142 :=[[15.8732060546875,-188.7220625,22.869189453125],[0.696320279376617,-0.571579290814731,-0.275420255163045,0.335527742350052],[0,0,0,0],[8.999999E+09,8.999999E+09,8.999999E+09,8.999999E+09,8.999999E+09,8.999999E+09]];
	LOCAL CONST Robtarget Tr_meulage_motif_1_P143 :=[[16.46945703125,-187.919265625,22.869208984375],[0.696320279376617,-0.571579290814731,-0.275420255163045,0.335527742350052],[0,0,0,0],[8.999999E+09,8.999999E+09,8.999999E+09,8.999999E+09,8.999999E+09,8.999999E+09]];
	LOCAL CONST Robtarget Tr_meulage_motif_1_P144 :=[[17.06570703125,-187.116453125,22.86923046875],[0.696320279376617,-0.571579290814731,-0.275420255163045,0.335527742350052],[0,0,0,0],[8.999999E+09,8.999999E+09,8.999999E+09,8.999999E+09,8.999999E+09,8.999999E+09]];
	LOCAL CONST Robtarget Tr_meulage_motif_1_P145 :=[[17.66195703125,-186.31365625,22.86925],[0.696320279376617,-0.571579290814731,-0.275420255163045,0.335527742350052],[0,0,0,0],[8.999999E+09,8.999999E+09,8.999999E+09,8.999999E+09,8.999999E+09,8.999999E+09]];
	LOCAL CONST Robtarget Tr_meulage_motif_1_P146 :=[[18.25820703125,-185.510859375,22.86926953125],[0.696320279376617,-0.571579290814731,-0.275420255163045,0.335527742350052],[0,0,0,0],[8.999999E+09,8.999999E+09,8.999999E+09,8.999999E+09,8.999999E+09,8.999999E+09]];
	LOCAL CONST Robtarget Tr_meulage_motif_1_P147 :=[[18.85445703125,-184.7080625,22.869291015625],[0.696320279376617,-0.571579290814731,-0.275420255163045,0.335527742350052],[0,0,0,0],[8.999999E+09,8.999999E+09,8.999999E+09,8.999999E+09,8.999999E+09,8.999999E+09]];
	LOCAL CONST Robtarget Tr_meulage_motif_1_P148 :=[[19.45070703125,-183.905265625,22.869310546875],[0.696320279376617,-0.571579290814731,-0.275420255163045,0.335527742350052],[0,0,0,0],[8.999999E+09,8.999999E+09,8.999999E+09,8.999999E+09,8.999999E+09,8.999999E+09]];
	LOCAL CONST Robtarget Tr_meulage_motif_1_P149 :=[[20.04695703125,-183.10246875,22.869330078125],[0.696320279376617,-0.571579290814731,-0.275420255163045,0.335527742350052],[0,0,0,0],[8.999999E+09,8.999999E+09,8.999999E+09,8.999999E+09,8.999999E+09,8.999999E+09]];
	LOCAL CONST Robtarget Tr_meulage_motif_1_P150 :=[[20.643208984375,-182.299671875,22.8693515625],[0.696320279376617,-0.571579290814731,-0.275420255163045,0.335527742350052],[0,0,0,0],[8.999999E+09,8.999999E+09,8.999999E+09,8.999999E+09,8.999999E+09,8.999999E+09]];
	LOCAL CONST Robtarget Tr_meulage_motif_1_P151 :=[[21.239458984375,-181.496875,22.86937109375],[0.696320279376617,-0.571579290814731,-0.275420255163045,0.335527742350052],[0,0,0,0],[8.999999E+09,8.999999E+09,8.999999E+09,8.999999E+09,8.999999E+09,8.999999E+09]];
	LOCAL CONST Robtarget Tr_meulage_motif_1_P152 :=[[21.835708984375,-180.694078125,22.869392578125],[0.696320279376617,-0.571579290814731,-0.275420255163045,0.335527742350052],[0,0,0,0],[8.999999E+09,8.999999E+09,8.999999E+09,8.999999E+09,8.999999E+09,8.999999E+09]];
	LOCAL CONST Robtarget Tr_meulage_motif_1_P153 :=[[22.431958984375,-179.891265625,22.869412109375],[0.696320279376617,-0.571579290814731,-0.275420255163045,0.335527742350052],[0,0,0,0],[8.999999E+09,8.999999E+09,8.999999E+09,8.999999E+09,8.999999E+09,8.999999E+09]];
	LOCAL CONST Robtarget Tr_meulage_motif_1_P154 :=[[23.028208984375,-179.08846875,22.869431640625],[0.696320279376617,-0.571579290814731,-0.275420255163045,0.335527742350052],[0,0,0,0],[8.999999E+09,8.999999E+09,8.999999E+09,8.999999E+09,8.999999E+09,8.999999E+09]];
	LOCAL CONST Robtarget Tr_meulage_motif_1_P155 :=[[23.624458984375,-178.285671875,22.869453125],[0.696320279376617,-0.571579290814731,-0.275420255163045,0.335527742350052],[0,0,0,0],[8.999999E+09,8.999999E+09,8.999999E+09,8.999999E+09,8.999999E+09,8.999999E+09]];
	LOCAL CONST Robtarget Tr_meulage_motif_1_P156 :=[[24.2207109375,-177.482875,22.86947265625],[0.696320279376617,-0.571579290814731,-0.275420255163045,0.335527742350052],[0,0,0,0],[8.999999E+09,8.999999E+09,8.999999E+09,8.999999E+09,8.999999E+09,8.999999E+09]];
	LOCAL CONST Robtarget Tr_meulage_motif_1_P157 :=[[24.8169609375,-176.680078125,22.8694921875],[0.696320279376617,-0.571579290814731,-0.275420255163045,0.335527742350052],[0,0,0,0],[8.999999E+09,8.999999E+09,8.999999E+09,8.999999E+09,8.999999E+09,8.999999E+09]];
	LOCAL CONST Robtarget Tr_meulage_motif_1_P158 :=[[25.4132109375,-175.87728125,22.869513671875],[0.696320279376617,-0.571579290814731,-0.275420255163045,0.335527742350052],[0,0,0,0],[8.999999E+09,8.999999E+09,8.999999E+09,8.999999E+09,8.999999E+09,8.999999E+09]];
	LOCAL CONST Robtarget Tr_meulage_motif_1_P159 :=[[26.0094609375,-175.074484375,22.869533203125],[0.696320279376617,-0.571579290814731,-0.275420255163045,0.335527742350052],[0,0,0,0],[8.999999E+09,8.999999E+09,8.999999E+09,8.999999E+09,8.999999E+09,8.999999E+09]];
	LOCAL CONST Robtarget Tr_meulage_motif_1_P160 :=[[26.6057109375,-174.2716875,22.8695546875],[0.696320279376617,-0.571579290814731,-0.275420255163045,0.335527742350052],[0,0,0,0],[8.999999E+09,8.999999E+09,8.999999E+09,8.999999E+09,8.999999E+09,8.999999E+09]];
	LOCAL CONST Robtarget Tr_meulage_motif_1_P161 :=[[27.2019609375,-173.468890625,22.86957421875],[0.696320279376617,-0.571579290814731,-0.275420255163045,0.335527742350052],[0,0,0,0],[8.999999E+09,8.999999E+09,8.999999E+09,8.999999E+09,8.999999E+09,8.999999E+09]];
	LOCAL CONST Robtarget Tr_meulage_motif_1_P162 :=[[27.7982109375,-172.666078125,22.86959375],[0.696320279376617,-0.571579290814731,-0.275420255163045,0.335527742350052],[0,0,0,0],[8.999999E+09,8.999999E+09,8.999999E+09,8.999999E+09,8.999999E+09,8.999999E+09]];
	LOCAL CONST Robtarget Tr_meulage_motif_1_P163 :=[[28.394462890625,-171.86328125,22.869615234375],[0.696320279376617,-0.571579290814731,-0.275420255163045,0.335527742350052],[0,0,0,0],[8.999999E+09,8.999999E+09,8.999999E+09,8.999999E+09,8.999999E+09,8.999999E+09]];
	LOCAL CONST Robtarget Tr_meulage_motif_1_P164 :=[[28.990712890625,-171.060484375,22.869634765625],[0.696320279376617,-0.571579290814731,-0.275420255163045,0.335527742350052],[0,0,0,0],[8.999999E+09,8.999999E+09,8.999999E+09,8.999999E+09,8.999999E+09,8.999999E+09]];
	LOCAL CONST Robtarget Tr_meulage_motif_1_P165 :=[[29.586962890625,-170.2576875,22.869654296875],[0.696320279376617,-0.571579290814731,-0.275420255163045,0.335527742350052],[0,0,0,0],[8.999999E+09,8.999999E+09,8.999999E+09,8.999999E+09,8.999999E+09,8.999999E+09]];
	LOCAL CONST Robtarget Tr_meulage_motif_1_P166 :=[[30.183212890625,-169.454890625,22.86967578125],[0.696320279376617,-0.571579290814731,-0.275420255163045,0.335527742350052],[0,0,0,0],[8.999999E+09,8.999999E+09,8.999999E+09,8.999999E+09,8.999999E+09,8.999999E+09]];
	LOCAL CONST Robtarget Tr_meulage_motif_1_P167 :=[[30.779462890625,-168.65209375,22.8696953125],[0.696320279376617,-0.571579290814731,-0.275420255163045,0.335527742350052],[0,0,0,0],[8.999999E+09,8.999999E+09,8.999999E+09,8.999999E+09,8.999999E+09,8.999999E+09]];
	LOCAL CONST Robtarget Tr_meulage_motif_1_P168 :=[[31.375712890625,-167.849296875,22.869716796875],[0.696320279376617,-0.571579290814731,-0.275420255163045,0.335527742350052],[0,0,0,0],[8.999999E+09,8.999999E+09,8.999999E+09,8.999999E+09,8.999999E+09,8.999999E+09]];
	LOCAL CONST Robtarget Tr_meulage_motif_1_P169 :=[[31.971962890625,-167.0465,22.869736328125],[0.696320279376617,-0.571579290814731,-0.275420255163045,0.335527742350052],[0,0,0,0],[8.999999E+09,8.999999E+09,8.999999E+09,8.999999E+09,8.999999E+09,8.999999E+09]];
	LOCAL CONST Robtarget Tr_meulage_motif_1_P170 :=[[32.56821484375,-166.243703125,22.869755859375],[0.696320279376617,-0.571579290814731,-0.275420255163045,0.335527742350052],[0,0,0,0],[8.999999E+09,8.999999E+09,8.999999E+09,8.999999E+09,8.999999E+09,8.999999E+09]];
	LOCAL CONST Robtarget Tr_meulage_motif_1_P171 :=[[33.16446484375,-165.440890625,22.86977734375],[0.696320279376617,-0.571579290814731,-0.275420255163045,0.335527742350052],[0,0,0,0],[8.999999E+09,8.999999E+09,8.999999E+09,8.999999E+09,8.999999E+09,8.999999E+09]];
	LOCAL CONST Robtarget Tr_meulage_motif_1_P172 :=[[33.76071484375,-164.63809375,22.869796875],[0.696320279376617,-0.571579290814731,-0.275420255163045,0.335527742350052],[0,0,0,0],[8.999999E+09,8.999999E+09,8.999999E+09,8.999999E+09,8.999999E+09,8.999999E+09]];
	LOCAL CONST Robtarget Tr_meulage_motif_1_P173 :=[[34.35696484375,-163.835296875,22.86981640625],[0.696320279376617,-0.571579290814731,-0.275420255163045,0.335527742350052],[0,0,0,0],[8.999999E+09,8.999999E+09,8.999999E+09,8.999999E+09,8.999999E+09,8.999999E+09]];
	LOCAL CONST Robtarget Tr_meulage_motif_1_P174 :=[[34.95321484375,-163.0325,22.869837890625],[0.696320279376617,-0.571579290814731,-0.275420255163045,0.335527742350052],[0,0,0,0],[8.999999E+09,8.999999E+09,8.999999E+09,8.999999E+09,8.999999E+09,8.999999E+09]];
	LOCAL CONST Robtarget Tr_meulage_motif_1_P175 :=[[35.54946484375,-162.229703125,22.869857421875],[0.696320279376617,-0.571579290814731,-0.275420255163045,0.335527742350052],[0,0,0,0],[8.999999E+09,8.999999E+09,8.999999E+09,8.999999E+09,8.999999E+09,8.999999E+09]];
	LOCAL CONST Robtarget Tr_meulage_motif_1_P176 :=[[36.14571484375,-161.42690625,22.86987890625],[0.696320279376617,-0.571579290814731,-0.275420255163045,0.335527742350052],[0,0,0,0],[8.999999E+09,8.999999E+09,8.999999E+09,8.999999E+09,8.999999E+09,8.999999E+09]];
	LOCAL CONST Robtarget Tr_meulage_motif_1_P177 :=[[36.74166015625,-160.633140625,22.759423828125],[0.696320279376617,-0.571579290814731,-0.275420255163045,0.335527742350052],[0,0,0,0],[8.999999E+09,8.999999E+09,8.999999E+09,8.999999E+09,8.999999E+09,8.999999E+09]];
	LOCAL CONST Robtarget Tr_meulage_motif_1_P178 :=[[37.31389453125,-159.879140625,22.548484375],[0.696320279376617,-0.571579290814731,-0.275420255163045,0.335527742350052],[0,0,0,0],[8.999999E+09,8.999999E+09,8.999999E+09,8.999999E+09,8.999999E+09,8.999999E+09]];
	LOCAL CONST Robtarget Tr_meulage_motif_1_P179 :=[[37.83247265625,-159.202109375,22.276951171875],[0.696320279376617,-0.571579290814731,-0.275420255163045,0.335527742350052],[0,0,0,0],[8.999999E+09,8.999999E+09,8.999999E+09,8.999999E+09,8.999999E+09,8.999999E+09]];
	LOCAL CONST Robtarget Tr_meulage_motif_1_P180 :=[[38.28992578125,-158.607703125,22.001328125],[0.696320279376617,-0.571579290814731,-0.275420255163045,0.335527742350052],[0,0,0,0],[8.999999E+09,8.999999E+09,8.999999E+09,8.999999E+09,8.999999E+09,8.999999E+09]];
	LOCAL CONST Robtarget Tr_meulage_motif_1_P181 :=[[38.9694296875,-157.74084375,21.385890625],[0.696320279376617,-0.571579290814731,-0.275420255163045,0.335527742350052],[0,0,0,0],[8.999999E+09,8.999999E+09,8.999999E+09,8.999999E+09,8.999999E+09,8.999999E+09]];
	LOCAL CONST Robtarget Tr_meulage_motif_1_P182 :=[[39.61155859375,-156.94234375,20.539171875],[0.696320279376617,-0.571579290814731,-0.275420255163045,0.335527742350052],[0,0,0,0],[8.999999E+09,8.999999E+09,8.999999E+09,8.999999E+09,8.999999E+09,8.999999E+09]];
	LOCAL CONST Robtarget Tr_meulage_motif_1_P183 :=[[40.15519140625,-156.29021875,19.516419921875],[0.696320279376617,-0.571579290814731,-0.275420255163045,0.335527742350052],[0,0,0,0],[8.999999E+09,8.999999E+09,8.999999E+09,8.999999E+09,8.999999E+09,8.999999E+09]];
	LOCAL CONST Robtarget Tr_meulage_motif_1_P184 :=[[40.48791796875,-155.929234375,18.40144921875],[0.696320279376617,-0.571579290814731,-0.275420255163045,0.335527742350052],[0,0,0,0],[8.999999E+09,8.999999E+09,8.999999E+09,8.999999E+09,8.999999E+09,8.999999E+09]];
	LOCAL CONST Robtarget Tr_meulage_motif_1_P185 :=[[40.53003125,-155.92678125,17.706232421875],[0.696320279376617,-0.571579290814731,-0.275420255163045,0.335527742350052],[0,0,0,0],[8.999999E+09,8.999999E+09,8.999999E+09,8.999999E+09,8.999999E+09,8.999999E+09]];
	LOCAL CONST Robtarget Tr_meulage_motif_1_P186 :=[[40.55471484375,-155.945109375,17.045697265625],[0.696320279376617,-0.571579290814731,-0.275420255163045,0.335527742350052],[0,0,0,0],[8.999999E+09,8.999999E+09,8.999999E+09,8.999999E+09,8.999999E+09,8.999999E+09]];
	LOCAL CONST Robtarget Tr_meulage_motif_1_P187 :=[[40.546671875,-156.00746875,16.38531640625],[0.696320279376617,-0.571579290814731,-0.275420255163045,0.335527742350052],[0,0,0,0],[8.999999E+09,8.999999E+09,8.999999E+09,8.999999E+09,8.999999E+09,8.999999E+09]];
	LOCAL CONST Robtarget Tr_meulage_motif_1_P188 :=[[40.290734375,-156.437953125,15.284748046875],[0.696320279376617,-0.571579290814731,-0.275420255163045,0.335527742350052],[0,0,0,0],[8.999999E+09,8.999999E+09,8.999999E+09,8.999999E+09,8.999999E+09,8.999999E+09]];
	LOCAL CONST Robtarget Tr_meulage_motif_1_P189 :=[[39.81754296875,-157.15353125,14.279193359375],[0.696320279376617,-0.571579290814731,-0.275420255163045,0.335527742350052],[0,0,0,0],[8.999999E+09,8.999999E+09,8.999999E+09,8.999999E+09,8.999999E+09,8.999999E+09]];
	LOCAL CONST Robtarget Tr_meulage_motif_1_P190 :=[[39.23827734375,-157.998078125,13.451193359375],[0.696320279376617,-0.571579290814731,-0.275420255163045,0.335527742350052],[0,0,0,0],[8.999999E+09,8.999999E+09,8.999999E+09,8.999999E+09,8.999999E+09,8.999999E+09]];
	LOCAL CONST Robtarget Tr_meulage_motif_1_P191 :=[[38.84337109375,-158.560640625,13.055857421875],[0.696320279376617,-0.571579290814731,-0.275420255163045,0.335527742350052],[0,0,0,0],[8.999999E+09,8.999999E+09,8.999999E+09,8.999999E+09,8.999999E+09,8.999999E+09]];
	LOCAL CONST Robtarget Tr_meulage_motif_1_P192 :=[[38.171015625,-159.50390625,12.5688291015625],[0.696320279376617,-0.571579290814731,-0.275420255163045,0.335527742350052],[0,0,0,0],[8.999999E+09,8.999999E+09,8.999999E+09,8.999999E+09,8.999999E+09,8.999999E+09]];
	LOCAL CONST Robtarget Tr_meulage_motif_1_P193 :=[[37.6770234375,-160.189609375,12.30500390625],[0.696320279376617,-0.571579290814731,-0.275420255163045,0.335527742350052],[0,0,0,0],[8.999999E+09,8.999999E+09,8.999999E+09,8.999999E+09,8.999999E+09,8.999999E+09]];
	LOCAL CONST Robtarget Tr_meulage_motif_1_P194 :=[[37.128953125,-160.943484375,12.1007373046875],[0.696320279376617,-0.571579290814731,-0.275420255163045,0.335527742350052],[0,0,0,0],[8.999999E+09,8.999999E+09,8.999999E+09,8.999999E+09,8.999999E+09,8.999999E+09]];
	LOCAL CONST Robtarget Tr_meulage_motif_1_P195 :=[[36.54774609375,-161.734484375,11.9922412109375],[0.696320279376617,-0.571579290814731,-0.275420255163045,0.335527742350052],[0,0,0,0],[8.999999E+09,8.999999E+09,8.999999E+09,8.999999E+09,8.999999E+09,8.999999E+09]];
	LOCAL CONST Robtarget Tr_meulage_motif_1_P196 :=[[35.96005859375,-162.534375,11.8817470703125],[0.696320279376617,-0.571579290814731,-0.275420255163045,0.335527742350052],[0,0,0,0],[8.999999E+09,8.999999E+09,8.999999E+09,8.999999E+09,8.999999E+09,8.999999E+09]];
	LOCAL CONST Robtarget Tr_meulage_motif_1_P197 :=[[35.36380859375,-163.337171875,11.8817265625],[0.696320279376617,-0.571579290814731,-0.275420255163045,0.335527742350052],[0,0,0,0],[8.999999E+09,8.999999E+09,8.999999E+09,8.999999E+09,8.999999E+09,8.999999E+09]];
	LOCAL CONST Robtarget Tr_meulage_motif_1_P198 :=[[34.76755859375,-164.139984375,11.8817060546875],[0.696320279376617,-0.571579290814731,-0.275420255163045,0.335527742350052],[0,0,0,0],[8.999999E+09,8.999999E+09,8.999999E+09,8.999999E+09,8.999999E+09,8.999999E+09]];
	LOCAL CONST Robtarget Tr_meulage_motif_1_P199 :=[[34.17130859375,-164.94278125,11.8816865234375],[0.696320279376617,-0.571579290814731,-0.275420255163045,0.335527742350052],[0,0,0,0],[8.999999E+09,8.999999E+09,8.999999E+09,8.999999E+09,8.999999E+09,8.999999E+09]];
	LOCAL CONST Robtarget Tr_meulage_motif_1_P200 :=[[33.57505859375,-165.745578125,11.881666015625],[0.696320279376617,-0.571579290814731,-0.275420255163045,0.335527742350052],[0,0,0,0],[8.999999E+09,8.999999E+09,8.999999E+09,8.999999E+09,8.999999E+09,8.999999E+09]];
	LOCAL CONST Robtarget Tr_meulage_motif_1_P201 :=[[32.97880859375,-166.548375,11.8816455078125],[0.696320279376617,-0.571579290814731,-0.275420255163045,0.335527742350052],[0,0,0,0],[8.999999E+09,8.999999E+09,8.999999E+09,8.999999E+09,8.999999E+09,8.999999E+09]];
	LOCAL CONST Robtarget Tr_meulage_motif_1_P202 :=[[32.38255859375,-167.351171875,11.881625],[0.696320279376617,-0.571579290814731,-0.275420255163045,0.335527742350052],[0,0,0,0],[8.999999E+09,8.999999E+09,8.999999E+09,8.999999E+09,8.999999E+09,8.999999E+09]];
	LOCAL CONST Robtarget Tr_meulage_motif_1_P203 :=[[31.78630859375,-168.15396875,11.88160546875],[0.696320279376617,-0.571579290814731,-0.275420255163045,0.335527742350052],[0,0,0,0],[8.999999E+09,8.999999E+09,8.999999E+09,8.999999E+09,8.999999E+09,8.999999E+09]];
	LOCAL CONST Robtarget Tr_meulage_motif_1_P204 :=[[31.19005859375,-168.956765625,11.8815849609375],[0.696320279376617,-0.571579290814731,-0.275420255163045,0.335527742350052],[0,0,0,0],[8.999999E+09,8.999999E+09,8.999999E+09,8.999999E+09,8.999999E+09,8.999999E+09]];
	LOCAL CONST Robtarget Tr_meulage_motif_1_P205 :=[[30.59380859375,-169.7595625,11.881564453125],[0.696320279376617,-0.571579290814731,-0.275420255163045,0.335527742350052],[0,0,0,0],[8.999999E+09,8.999999E+09,8.999999E+09,8.999999E+09,8.999999E+09,8.999999E+09]];
	LOCAL CONST Robtarget Tr_meulage_motif_1_P206 :=[[29.997556640625,-170.562359375,11.8815439453125],[0.696320279376617,-0.571579290814731,-0.275420255163045,0.335527742350052],[0,0,0,0],[8.999999E+09,8.999999E+09,8.999999E+09,8.999999E+09,8.999999E+09,8.999999E+09]];
	LOCAL CONST Robtarget Tr_meulage_motif_1_P207 :=[[29.401306640625,-171.365171875,11.8815244140625],[0.696320279376617,-0.571579290814731,-0.275420255163045,0.335527742350052],[0,0,0,0],[8.999999E+09,8.999999E+09,8.999999E+09,8.999999E+09,8.999999E+09,8.999999E+09]];
	LOCAL CONST Robtarget Tr_meulage_motif_1_P208 :=[[28.805056640625,-172.16796875,11.88150390625],[0.696320279376617,-0.571579290814731,-0.275420255163045,0.335527742350052],[0,0,0,0],[8.999999E+09,8.999999E+09,8.999999E+09,8.999999E+09,8.999999E+09,8.999999E+09]];
	LOCAL CONST Robtarget Tr_meulage_motif_1_P209 :=[[28.208806640625,-172.970765625,11.8814833984375],[0.696320279376617,-0.571579290814731,-0.275420255163045,0.335527742350052],[0,0,0,0],[8.999999E+09,8.999999E+09,8.999999E+09,8.999999E+09,8.999999E+09,8.999999E+09]];
	LOCAL CONST Robtarget Tr_meulage_motif_1_P210 :=[[27.612556640625,-173.7735625,11.881462890625],[0.696320279376617,-0.571579290814731,-0.275420255163045,0.335527742350052],[0,0,0,0],[8.999999E+09,8.999999E+09,8.999999E+09,8.999999E+09,8.999999E+09,8.999999E+09]];
	LOCAL CONST Robtarget Tr_meulage_motif_1_P211 :=[[27.016306640625,-174.576359375,11.881443359375],[0.696320279376617,-0.571579290814731,-0.275420255163045,0.335527742350052],[0,0,0,0],[8.999999E+09,8.999999E+09,8.999999E+09,8.999999E+09,8.999999E+09,8.999999E+09]];
	LOCAL CONST Robtarget Tr_meulage_motif_1_P212 :=[[26.420056640625,-175.37915625,11.8814228515625],[0.696320279376617,-0.571579290814731,-0.275420255163045,0.335527742350052],[0,0,0,0],[8.999999E+09,8.999999E+09,8.999999E+09,8.999999E+09,8.999999E+09,8.999999E+09]];
	LOCAL CONST Robtarget Tr_meulage_motif_1_P213 :=[[25.8238046875,-176.181953125,11.88140234375],[0.696320279376617,-0.571579290814731,-0.275420255163045,0.335527742350052],[0,0,0,0],[8.999999E+09,8.999999E+09,8.999999E+09,8.999999E+09,8.999999E+09,8.999999E+09]];
	LOCAL CONST Robtarget Tr_meulage_motif_1_P214 :=[[25.2275546875,-176.98475,11.8813818359375],[0.696320279376617,-0.571579290814731,-0.275420255163045,0.335527742350052],[0,0,0,0],[8.999999E+09,8.999999E+09,8.999999E+09,8.999999E+09,8.999999E+09,8.999999E+09]];
	LOCAL CONST Robtarget Tr_meulage_motif_1_P215 :=[[24.6313046875,-177.787546875,11.8813623046875],[0.696320279376617,-0.571579290814731,-0.275420255163045,0.335527742350052],[0,0,0,0],[8.999999E+09,8.999999E+09,8.999999E+09,8.999999E+09,8.999999E+09,8.999999E+09]];
	LOCAL CONST Robtarget Tr_meulage_motif_1_P216 :=[[24.0350546875,-178.590359375,11.881341796875],[0.696320279376617,-0.571579290814731,-0.275420255163045,0.335527742350052],[0,0,0,0],[8.999999E+09,8.999999E+09,8.999999E+09,8.999999E+09,8.999999E+09,8.999999E+09]];
	LOCAL CONST Robtarget Tr_meulage_motif_1_P217 :=[[23.4388046875,-179.39315625,11.8813212890625],[0.696320279376617,-0.571579290814731,-0.275420255163045,0.335527742350052],[0,0,0,0],[8.999999E+09,8.999999E+09,8.999999E+09,8.999999E+09,8.999999E+09,8.999999E+09]];
	LOCAL CONST Robtarget Tr_meulage_motif_1_P218 :=[[22.8425546875,-180.195953125,11.88130078125],[0.696320279376617,-0.571579290814731,-0.275420255163045,0.335527742350052],[0,0,0,0],[8.999999E+09,8.999999E+09,8.999999E+09,8.999999E+09,8.999999E+09,8.999999E+09]];
	LOCAL CONST Robtarget Tr_meulage_motif_1_P219 :=[[22.246302734375,-180.99875,11.88128125],[0.696320279376617,-0.571579290814731,-0.275420255163045,0.335527742350052],[0,0,0,0],[8.999999E+09,8.999999E+09,8.999999E+09,8.999999E+09,8.999999E+09,8.999999E+09]];
	LOCAL CONST Robtarget Tr_meulage_motif_1_P220 :=[[21.650052734375,-181.801546875,11.8812607421875],[0.696320279376617,-0.571579290814731,-0.275420255163045,0.335527742350052],[0,0,0,0],[8.999999E+09,8.999999E+09,8.999999E+09,8.999999E+09,8.999999E+09,8.999999E+09]];
	LOCAL CONST Robtarget Tr_meulage_motif_1_P221 :=[[21.053802734375,-182.60434375,11.881240234375],[0.696320279376617,-0.571579290814731,-0.275420255163045,0.335527742350052],[0,0,0,0],[8.999999E+09,8.999999E+09,8.999999E+09,8.999999E+09,8.999999E+09,8.999999E+09]];
	LOCAL CONST Robtarget Tr_meulage_motif_1_P222 :=[[20.457552734375,-183.407140625,11.8812197265625],[0.696320279376617,-0.571579290814731,-0.275420255163045,0.335527742350052],[0,0,0,0],[8.999999E+09,8.999999E+09,8.999999E+09,8.999999E+09,8.999999E+09,8.999999E+09]];
	LOCAL CONST Robtarget Tr_meulage_motif_1_P223 :=[[19.861302734375,-184.2099375,11.8812001953125],[0.696320279376617,-0.571579290814731,-0.275420255163045,0.335527742350052],[0,0,0,0],[8.999999E+09,8.999999E+09,8.999999E+09,8.999999E+09,8.999999E+09,8.999999E+09]];
	LOCAL CONST Robtarget Tr_meulage_motif_1_P224 :=[[19.265052734375,-185.012734375,11.8811796875],[0.696320279376617,-0.571579290814731,-0.275420255163045,0.335527742350052],[0,0,0,0],[8.999999E+09,8.999999E+09,8.999999E+09,8.999999E+09,8.999999E+09,8.999999E+09]];
	LOCAL CONST Robtarget Tr_meulage_motif_1_P225 :=[[18.668802734375,-185.815546875,11.8811591796875],[0.696320279376617,-0.571579290814731,-0.275420255163045,0.335527742350052],[0,0,0,0],[8.999999E+09,8.999999E+09,8.999999E+09,8.999999E+09,8.999999E+09,8.999999E+09]];
	LOCAL CONST Robtarget Tr_meulage_motif_1_P226 :=[[18.07255078125,-186.61834375,11.881138671875],[0.696320279376617,-0.571579290814731,-0.275420255163045,0.335527742350052],[0,0,0,0],[8.999999E+09,8.999999E+09,8.999999E+09,8.999999E+09,8.999999E+09,8.999999E+09]];
	LOCAL CONST Robtarget Tr_meulage_motif_1_P227 :=[[17.47630078125,-187.421140625,11.881119140625],[0.696320279376617,-0.571579290814731,-0.275420255163045,0.335527742350052],[0,0,0,0],[8.999999E+09,8.999999E+09,8.999999E+09,8.999999E+09,8.999999E+09,8.999999E+09]];
	LOCAL CONST Robtarget Tr_meulage_motif_1_P228 :=[[16.88005078125,-188.2239375,11.8810986328125],[0.696320279376617,-0.571579290814731,-0.275420255163045,0.335527742350052],[0,0,0,0],[8.999999E+09,8.999999E+09,8.999999E+09,8.999999E+09,8.999999E+09,8.999999E+09]];
	LOCAL CONST Robtarget Tr_meulage_motif_1_P229 :=[[16.28380078125,-189.026734375,11.881078125],[0.696320279376617,-0.571579290814731,-0.275420255163045,0.335527742350052],[0,0,0,0],[8.999999E+09,8.999999E+09,8.999999E+09,8.999999E+09,8.999999E+09,8.999999E+09]];
	LOCAL CONST Robtarget Tr_meulage_motif_1_P230 :=[[15.68755078125,-189.82953125,11.8810576171875],[0.696320279376617,-0.571579290814731,-0.275420255163045,0.335527742350052],[0,0,0,0],[8.999999E+09,8.999999E+09,8.999999E+09,8.999999E+09,8.999999E+09,8.999999E+09]];
	LOCAL CONST Robtarget Tr_meulage_motif_1_P231 :=[[15.0912998046875,-190.632328125,11.8810380859375],[0.696320279376617,-0.571579290814731,-0.275420255163045,0.335527742350052],[0,0,0,0],[8.999999E+09,8.999999E+09,8.999999E+09,8.999999E+09,8.999999E+09,8.999999E+09]];
	LOCAL CONST Robtarget Tr_meulage_motif_1_P232 :=[[14.4950498046875,-191.435125,11.881017578125],[0.696320279376617,-0.571579290814731,-0.275420255163045,0.335527742350052],[0,0,0,0],[8.999999E+09,8.999999E+09,8.999999E+09,8.999999E+09,8.999999E+09,8.999999E+09]];
	LOCAL CONST Robtarget Tr_meulage_motif_1_P233 :=[[13.8987998046875,-192.237921875,11.8809970703125],[0.696320279376617,-0.571579290814731,-0.275420255163045,0.335527742350052],[0,0,0,0],[8.999999E+09,8.999999E+09,8.999999E+09,8.999999E+09,8.999999E+09,8.999999E+09]];
	LOCAL CONST Robtarget Tr_meulage_motif_1_P234 :=[[13.302548828125,-193.040734375,11.8809765625],[0.696320279376617,-0.571579290814731,-0.275420255163045,0.335527742350052],[0,0,0,0],[8.999999E+09,8.999999E+09,8.999999E+09,8.999999E+09,8.999999E+09,8.999999E+09]];
	LOCAL CONST Robtarget Tr_meulage_motif_1_P235 :=[[12.706298828125,-193.84353125,11.88095703125],[0.696320279376617,-0.571579290814731,-0.275420255163045,0.335527742350052],[0,0,0,0],[8.999999E+09,8.999999E+09,8.999999E+09,8.999999E+09,8.999999E+09,8.999999E+09]];
	LOCAL CONST Robtarget Tr_meulage_motif_1_P236 :=[[12.110048828125,-194.646328125,11.8809365234375],[0.696320279376617,-0.571579290814731,-0.275420255163045,0.335527742350052],[0,0,0,0],[8.999999E+09,8.999999E+09,8.999999E+09,8.999999E+09,8.999999E+09,8.999999E+09]];
	LOCAL CONST Robtarget Tr_meulage_motif_1_P237 :=[[11.513798828125,-195.449125,11.880916015625],[0.696320279376617,-0.571579290814731,-0.275420255163045,0.335527742350052],[0,0,0,0],[8.999999E+09,8.999999E+09,8.999999E+09,8.999999E+09,8.999999E+09,8.999999E+09]];
	LOCAL CONST Robtarget Tr_meulage_motif_1_P238 :=[[10.9175478515625,-196.251921875,11.8808955078125],[0.696320279376617,-0.571579290814731,-0.275420255163045,0.335527742350052],[0,0,0,0],[8.999999E+09,8.999999E+09,8.999999E+09,8.999999E+09,8.999999E+09,8.999999E+09]];
	LOCAL CONST Robtarget Tr_meulage_motif_1_P239 :=[[10.3212978515625,-197.05471875,11.8808759765625],[0.696320279376617,-0.571579290814731,-0.275420255163045,0.335527742350052],[0,0,0,0],[8.999999E+09,8.999999E+09,8.999999E+09,8.999999E+09,8.999999E+09,8.999999E+09]];
	LOCAL CONST Robtarget Tr_meulage_motif_1_P240 :=[[9.7336103515625,-197.854609375,11.770380859375],[0.696320279376617,-0.571579290814731,-0.275420255163045,0.335527742350052],[0,0,0,0],[8.999999E+09,8.999999E+09,8.999999E+09,8.999999E+09,8.999999E+09,8.999999E+09]];
	LOCAL CONST Robtarget Tr_meulage_motif_1_P241 :=[[9.177142578125,-198.6203125,11.55940234375],[0.696320279376617,-0.571579290814731,-0.275420255163045,0.335527742350052],[0,0,0,0],[8.999999E+09,8.999999E+09,8.999999E+09,8.999999E+09,8.999999E+09,8.999999E+09]];
	LOCAL CONST Robtarget Tr_meulage_motif_1_P242 :=[[8.67885546875,-199.31240625,11.2878359375],[0.696320279376617,-0.571579290814731,-0.275420255163045,0.335527742350052],[0,0,0,0],[8.999999E+09,8.999999E+09,8.999999E+09,8.999999E+09,8.999999E+09,8.999999E+09]];
	LOCAL CONST Robtarget Tr_meulage_motif_1_P243 :=[[8.2659755859375,-199.892015625,10.9840087890625],[0.696320279376617,-0.571579290814731,-0.275420255163045,0.335527742350052],[0,0,0,0],[8.999999E+09,8.999999E+09,8.999999E+09,8.999999E+09,8.999999E+09,8.999999E+09]];
	LOCAL CONST Robtarget Tr_meulage_motif_1_P244 :=[[7.67390380859375,-200.74084375,10.3221728515625],[0.696320279376617,-0.571579290814731,-0.275420255163045,0.335527742350052],[0,0,0,0],[8.999999E+09,8.999999E+09,8.999999E+09,8.999999E+09,8.999999E+09,8.999999E+09]];
	LOCAL CONST Robtarget Tr_meulage_motif_1_P245 :=[[7.16979052734375,-201.489890625,9.4211767578125],[0.696320279376617,-0.571579290814731,-0.275420255163045,0.335527742350052],[0,0,0,0],[8.999999E+09,8.999999E+09,8.999999E+09,8.999999E+09,8.999999E+09,8.999999E+09]];
	LOCAL CONST Robtarget Tr_meulage_motif_1_P246 :=[[6.889859375,-201.94834375,8.3762802734375],[0.696320279376617,-0.571579290814731,-0.275420255163045,0.335527742350052],[0,0,0,0],[8.999999E+09,8.999999E+09,8.999999E+09,8.999999E+09,8.999999E+09,8.999999E+09]];
	LOCAL CONST Robtarget Tr_meulage_motif_1_P247 :=[[6.80556005859375,-202.115875,7.68379150390625],[0.696320279376617,-0.571579290814731,-0.275420255163045,0.335527742350052],[0,0,0,0],[8.999999E+09,8.999999E+09,8.999999E+09,8.999999E+09,8.999999E+09,8.999999E+09]];
	LOCAL CONST Robtarget Tr_meulage_motif_1_P248 :=[[6.79623486328125,-202.18846875,6.91462255859375],[0.696320279376617,-0.571579290814731,-0.275420255163045,0.335527742350052],[0,0,0,0],[8.999999E+09,8.999999E+09,8.999999E+09,8.999999E+09,8.999999E+09,8.999999E+09]];
	LOCAL CONST Robtarget Tr_meulage_motif_1_P249 :=[[6.8648828125,-202.156046875,6.1455966796875],[0.696320279376617,-0.571579290814731,-0.275420255163045,0.335527742350052],[0,0,0,0],[8.999999E+09,8.999999E+09,8.999999E+09,8.999999E+09,8.999999E+09,8.999999E+09]];
	LOCAL CONST Robtarget Tr_meulage_motif_1_P250 :=[[7.15643310546875,-201.849890625,5.03855322265625],[0.696320279376617,-0.571579290814731,-0.275420255163045,0.335527742350052],[0,0,0,0],[8.999999E+09,8.999999E+09,8.999999E+09,8.999999E+09,8.999999E+09,8.999999E+09]];
	LOCAL CONST Robtarget Tr_meulage_motif_1_P251 :=[[7.42532861328125,-201.533515625,4.4535068359375],[0.696320279376617,-0.571579290814731,-0.275420255163045,0.335527742350052],[0,0,0,0],[8.999999E+09,8.999999E+09,8.999999E+09,8.999999E+09,8.999999E+09,8.999999E+09]];
	LOCAL CONST Robtarget Tr_meulage_motif_1_P252 :=[[7.98739208984375,-200.845890625,3.56732763671875],[0.696320279376617,-0.571579290814731,-0.275420255163045,0.335527742350052],[0,0,0,0],[8.999999E+09,8.999999E+09,8.999999E+09,8.999999E+09,8.999999E+09,8.999999E+09]];
	LOCAL CONST Robtarget Tr_meulage_motif_1_P253 :=[[8.352072265625,-200.3871875,3.153505859375],[0.696320279376617,-0.571579290814731,-0.275420255163045,0.335527742350052],[0,0,0,0],[8.999999E+09,8.999999E+09,8.999999E+09,8.999999E+09,8.999999E+09,8.999999E+09]];
	LOCAL CONST Robtarget Tr_meulage_motif_1_P254 :=[[9.0389345703125,-199.504796875,2.60999169921875],[0.696320279376617,-0.571579290814731,-0.275420255163045,0.335527742350052],[0,0,0,0],[8.999999E+09,8.999999E+09,8.999999E+09,8.999999E+09,8.999999E+09,8.999999E+09]];
	LOCAL CONST Robtarget Tr_meulage_motif_1_P255 :=[[9.542224609375,-198.850203125,2.31482788085937],[0.696320279376617,-0.571579290814731,-0.275420255163045,0.335527742350052],[0,0,0,0],[8.999999E+09,8.999999E+09,8.999999E+09,8.999999E+09,8.999999E+09,8.999999E+09]];
	LOCAL CONST Robtarget Tr_meulage_motif_1_P256 :=[[10.1055634765625,-198.10765625,2.11058325195313],[0.696320279376617,-0.571579290814731,-0.275420255163045,0.335527742350052],[0,0,0,0],[8.999999E+09,8.999999E+09,8.999999E+09,8.999999E+09,8.999999E+09,8.999999E+09]];
	LOCAL CONST Robtarget Tr_meulage_motif_1_P257 :=[[10.6948720703125,-197.322671875,2.00217370605469],[0.696320279376617,-0.571579290814731,-0.275420255163045,0.335527742350052],[0,0,0,0],[8.999999E+09,8.999999E+09,8.999999E+09,8.999999E+09,8.999999E+09,8.999999E+09]];
	LOCAL CONST Robtarget Tr_meulage_motif_1_P258 :=[[11.29081640625,-196.52890625,1.89170397949219],[0.696320279376617,-0.571579290814731,-0.275420255163045,0.335527742350052],[0,0,0,0],[8.999999E+09,8.999999E+09,8.999999E+09,8.999999E+09,8.999999E+09,8.999999E+09]];
	LOCAL CONST Robtarget Tr_meulage_motif_1_P259 :=[[11.88706640625,-195.726109375,1.89172424316406],[0.696320279376617,-0.571579290814731,-0.275420255163045,0.335527742350052],[0,0,0,0],[8.999999E+09,8.999999E+09,8.999999E+09,8.999999E+09,8.999999E+09,8.999999E+09]];
	LOCAL CONST Robtarget Tr_meulage_motif_1_P260 :=[[12.48331640625,-194.923296875,1.89174450683594],[0.696320279376617,-0.571579290814731,-0.275420255163045,0.335527742350052],[0,0,0,0],[8.999999E+09,8.999999E+09,8.999999E+09,8.999999E+09,8.999999E+09,8.999999E+09]];
	LOCAL CONST Robtarget Tr_meulage_motif_1_P261 :=[[13.0795673828125,-194.1205,1.89176477050781],[0.696320279376617,-0.571579290814731,-0.275420255163045,0.335527742350052],[0,0,0,0],[8.999999E+09,8.999999E+09,8.999999E+09,8.999999E+09,8.999999E+09,8.999999E+09]];
	LOCAL CONST Robtarget Tr_meulage_motif_1_P262 :=[[13.6758173828125,-193.317703125,1.89178503417969],[0.696320279376617,-0.571579290814731,-0.275420255163045,0.335527742350052],[0,0,0,0],[8.999999E+09,8.999999E+09,8.999999E+09,8.999999E+09,8.999999E+09,8.999999E+09]];
	LOCAL CONST Robtarget Tr_meulage_motif_1_P263 :=[[14.2720673828125,-192.51490625,1.89180529785156],[0.696320279376617,-0.571579290814731,-0.275420255163045,0.335527742350052],[0,0,0,0],[8.999999E+09,8.999999E+09,8.999999E+09,8.999999E+09,8.999999E+09,8.999999E+09]];
	LOCAL CONST Robtarget Tr_meulage_motif_1_P264 :=[[14.8683173828125,-191.712109375,1.89182556152344],[0.696320279376617,-0.571579290814731,-0.275420255163045,0.335527742350052],[0,0,0,0],[8.999999E+09,8.999999E+09,8.999999E+09,8.999999E+09,8.999999E+09,8.999999E+09]];
	LOCAL CONST Robtarget Tr_meulage_motif_1_P265 :=[[15.464568359375,-190.9093125,1.89184582519531],[0.696320279376617,-0.571579290814731,-0.275420255163045,0.335527742350052],[0,0,0,0],[8.999999E+09,8.999999E+09,8.999999E+09,8.999999E+09,8.999999E+09,8.999999E+09]];
	LOCAL CONST Robtarget Tr_meulage_motif_1_P266 :=[[16.060818359375,-190.106515625,1.89186608886719],[0.696320279376617,-0.571579290814731,-0.275420255163045,0.335527742350052],[0,0,0,0],[8.999999E+09,8.999999E+09,8.999999E+09,8.999999E+09,8.999999E+09,8.999999E+09]];
	LOCAL CONST Robtarget Tr_meulage_motif_1_P267 :=[[16.657068359375,-189.30371875,1.89188635253906],[0.696320279376617,-0.571579290814731,-0.275420255163045,0.335527742350052],[0,0,0,0],[8.999999E+09,8.999999E+09,8.999999E+09,8.999999E+09,8.999999E+09,8.999999E+09]];
	LOCAL CONST Robtarget Tr_meulage_motif_1_P268 :=[[17.253318359375,-188.500921875,1.89190661621094],[0.696320279376617,-0.571579290814731,-0.275420255163045,0.335527742350052],[0,0,0,0],[8.999999E+09,8.999999E+09,8.999999E+09,8.999999E+09,8.999999E+09,8.999999E+09]];
	LOCAL CONST Robtarget Tr_meulage_motif_1_P269 :=[[17.849568359375,-187.698109375,1.89192687988281],[0.696320279376617,-0.571579290814731,-0.275420255163045,0.335527742350052],[0,0,0,0],[8.999999E+09,8.999999E+09,8.999999E+09,8.999999E+09,8.999999E+09,8.999999E+09]];
	LOCAL CONST Robtarget Tr_meulage_motif_1_P270 :=[[18.4458203125,-186.8953125,1.89194714355469],[0.696320279376617,-0.571579290814731,-0.275420255163045,0.335527742350052],[0,0,0,0],[8.999999E+09,8.999999E+09,8.999999E+09,8.999999E+09,8.999999E+09,8.999999E+09]];
	LOCAL CONST Robtarget Tr_meulage_motif_1_P271 :=[[19.0420703125,-186.092515625,1.89196740722656],[0.696320279376617,-0.571579290814731,-0.275420255163045,0.335527742350052],[0,0,0,0],[8.999999E+09,8.999999E+09,8.999999E+09,8.999999E+09,8.999999E+09,8.999999E+09]];
	LOCAL CONST Robtarget Tr_meulage_motif_1_P272 :=[[19.6383203125,-185.28971875,1.89198767089844],[0.696320279376617,-0.571579290814731,-0.275420255163045,0.335527742350052],[0,0,0,0],[8.999999E+09,8.999999E+09,8.999999E+09,8.999999E+09,8.999999E+09,8.999999E+09]];
	LOCAL CONST Robtarget Tr_meulage_motif_1_P273 :=[[20.2345703125,-184.486921875,1.89200793457031],[0.696320279376617,-0.571579290814731,-0.275420255163045,0.335527742350052],[0,0,0,0],[8.999999E+09,8.999999E+09,8.999999E+09,8.999999E+09,8.999999E+09,8.999999E+09]];
	LOCAL CONST Robtarget Tr_meulage_motif_1_P274 :=[[20.8308203125,-183.684125,1.89202819824219],[0.696320279376617,-0.571579290814731,-0.275420255163045,0.335527742350052],[0,0,0,0],[8.999999E+09,8.999999E+09,8.999999E+09,8.999999E+09,8.999999E+09,8.999999E+09]];
	LOCAL CONST Robtarget Tr_meulage_motif_1_P275 :=[[21.4270703125,-182.881328125,1.89204846191406],[0.696320279376617,-0.571579290814731,-0.275420255163045,0.335527742350052],[0,0,0,0],[8.999999E+09,8.999999E+09,8.999999E+09,8.999999E+09,8.999999E+09,8.999999E+09]];
	LOCAL CONST Robtarget Tr_meulage_motif_1_P276 :=[[22.023322265625,-182.07853125,1.89206872558594],[0.696320279376617,-0.571579290814731,-0.275420255163045,0.335527742350052],[0,0,0,0],[8.999999E+09,8.999999E+09,8.999999E+09,8.999999E+09,8.999999E+09,8.999999E+09]];
	LOCAL CONST Robtarget Tr_meulage_motif_1_P277 :=[[22.619572265625,-181.275734375,1.89208898925781],[0.696320279376617,-0.571579290814731,-0.275420255163045,0.335527742350052],[0,0,0,0],[8.999999E+09,8.999999E+09,8.999999E+09,8.999999E+09,8.999999E+09,8.999999E+09]];
	LOCAL CONST Robtarget Tr_meulage_motif_1_P278 :=[[23.215822265625,-180.472921875,1.89210925292969],[0.696320279376617,-0.571579290814731,-0.275420255163045,0.335527742350052],[0,0,0,0],[8.999999E+09,8.999999E+09,8.999999E+09,8.999999E+09,8.999999E+09,8.999999E+09]];
	LOCAL CONST Robtarget Tr_meulage_motif_1_P279 :=[[23.812072265625,-179.670125,1.89212951660156],[0.696320279376617,-0.571579290814731,-0.275420255163045,0.335527742350052],[0,0,0,0],[8.999999E+09,8.999999E+09,8.999999E+09,8.999999E+09,8.999999E+09,8.999999E+09]];
	LOCAL CONST Robtarget Tr_meulage_motif_1_P280 :=[[24.408322265625,-178.867328125,1.89214978027344],[0.696320279376617,-0.571579290814731,-0.275420255163045,0.335527742350052],[0,0,0,0],[8.999999E+09,8.999999E+09,8.999999E+09,8.999999E+09,8.999999E+09,8.999999E+09]];
	LOCAL CONST Robtarget Tr_meulage_motif_1_P281 :=[[25.004572265625,-178.06453125,1.89217004394531],[0.696320279376617,-0.571579290814731,-0.275420255163045,0.335527742350052],[0,0,0,0],[8.999999E+09,8.999999E+09,8.999999E+09,8.999999E+09,8.999999E+09,8.999999E+09]];
	LOCAL CONST Robtarget Tr_meulage_motif_1_P282 :=[[25.600822265625,-177.261734375,1.89219030761719],[0.696320279376617,-0.571579290814731,-0.275420255163045,0.335527742350052],[0,0,0,0],[8.999999E+09,8.999999E+09,8.999999E+09,8.999999E+09,8.999999E+09,8.999999E+09]];
	LOCAL CONST Robtarget Tr_meulage_motif_1_P283 :=[[26.19707421875,-176.4589375,1.89221057128906],[0.696320279376617,-0.571579290814731,-0.275420255163045,0.335527742350052],[0,0,0,0],[8.999999E+09,8.999999E+09,8.999999E+09,8.999999E+09,8.999999E+09,8.999999E+09]];
	LOCAL CONST Robtarget Tr_meulage_motif_1_P284 :=[[26.79332421875,-175.656140625,1.89223083496094],[0.696320279376617,-0.571579290814731,-0.275420255163045,0.335527742350052],[0,0,0,0],[8.999999E+09,8.999999E+09,8.999999E+09,8.999999E+09,8.999999E+09,8.999999E+09]];
	LOCAL CONST Robtarget Tr_meulage_motif_1_P285 :=[[27.38957421875,-174.85334375,1.89225109863281],[0.696320279376617,-0.571579290814731,-0.275420255163045,0.335527742350052],[0,0,0,0],[8.999999E+09,8.999999E+09,8.999999E+09,8.999999E+09,8.999999E+09,8.999999E+09]];
	LOCAL CONST Robtarget Tr_meulage_motif_1_P286 :=[[27.98582421875,-174.050546875,1.89227136230469],[0.696320279376617,-0.571579290814731,-0.275420255163045,0.335527742350052],[0,0,0,0],[8.999999E+09,8.999999E+09,8.999999E+09,8.999999E+09,8.999999E+09,8.999999E+09]];
	LOCAL CONST Robtarget Tr_meulage_motif_1_P287 :=[[28.58207421875,-173.247734375,1.89229162597656],[0.696320279376617,-0.571579290814731,-0.275420255163045,0.335527742350052],[0,0,0,0],[8.999999E+09,8.999999E+09,8.999999E+09,8.999999E+09,8.999999E+09,8.999999E+09]];
	LOCAL CONST Robtarget Tr_meulage_motif_1_P288 :=[[29.17832421875,-172.4449375,1.89231188964844],[0.696320279376617,-0.571579290814731,-0.275420255163045,0.335527742350052],[0,0,0,0],[8.999999E+09,8.999999E+09,8.999999E+09,8.999999E+09,8.999999E+09,8.999999E+09]];
	LOCAL CONST Robtarget Tr_meulage_motif_1_P289 :=[[29.77457421875,-171.642140625,1.89233215332031],[0.696320279376617,-0.571579290814731,-0.275420255163045,0.335527742350052],[0,0,0,0],[8.999999E+09,8.999999E+09,8.999999E+09,8.999999E+09,8.999999E+09,8.999999E+09]];
	LOCAL CONST Robtarget Tr_meulage_motif_1_P290 :=[[30.370826171875,-170.83934375,1.89235241699219],[0.696320279376617,-0.571579290814731,-0.275420255163045,0.335527742350052],[0,0,0,0],[8.999999E+09,8.999999E+09,8.999999E+09,8.999999E+09,8.999999E+09,8.999999E+09]];
	LOCAL CONST Robtarget Tr_meulage_motif_1_P291 :=[[30.967076171875,-170.036546875,1.89237268066406],[0.696320279376617,-0.571579290814731,-0.275420255163045,0.335527742350052],[0,0,0,0],[8.999999E+09,8.999999E+09,8.999999E+09,8.999999E+09,8.999999E+09,8.999999E+09]];
	LOCAL CONST Robtarget Tr_meulage_motif_1_P292 :=[[31.563326171875,-169.23375,1.89239294433594],[0.696320279376617,-0.571579290814731,-0.275420255163045,0.335527742350052],[0,0,0,0],[8.999999E+09,8.999999E+09,8.999999E+09,8.999999E+09,8.999999E+09,8.999999E+09]];
	LOCAL CONST Robtarget Tr_meulage_motif_1_P293 :=[[32.159576171875,-168.430953125,1.89241320800781],[0.696320279376617,-0.571579290814731,-0.275420255163045,0.335527742350052],[0,0,0,0],[8.999999E+09,8.999999E+09,8.999999E+09,8.999999E+09,8.999999E+09,8.999999E+09]];
	LOCAL CONST Robtarget Tr_meulage_motif_1_P294 :=[[32.755826171875,-167.62815625,1.89243347167969],[0.696320279376617,-0.571579290814731,-0.275420255163045,0.335527742350052],[0,0,0,0],[8.999999E+09,8.999999E+09,8.999999E+09,8.999999E+09,8.999999E+09,8.999999E+09]];
	LOCAL CONST Robtarget Tr_meulage_motif_1_P295 :=[[33.352078125,-166.825359375,1.89245373535156],[0.696320279376617,-0.571579290814731,-0.275420255163045,0.335527742350052],[0,0,0,0],[8.999999E+09,8.999999E+09,8.999999E+09,8.999999E+09,8.999999E+09,8.999999E+09]];
	LOCAL CONST Robtarget Tr_meulage_motif_1_P296 :=[[33.948328125,-166.022546875,1.89247399902344],[0.696320279376617,-0.571579290814731,-0.275420255163045,0.335527742350052],[0,0,0,0],[8.999999E+09,8.999999E+09,8.999999E+09,8.999999E+09,8.999999E+09,8.999999E+09]];
	LOCAL CONST Robtarget Tr_meulage_motif_1_P297 :=[[34.544578125,-165.21975,1.89249426269531],[0.696320279376617,-0.571579290814731,-0.275420255163045,0.335527742350052],[0,0,0,0],[8.999999E+09,8.999999E+09,8.999999E+09,8.999999E+09,8.999999E+09,8.999999E+09]];
	LOCAL CONST Robtarget Tr_meulage_motif_1_P298 :=[[35.140828125,-164.416953125,1.89251452636719],[0.696320279376617,-0.571579290814731,-0.275420255163045,0.335527742350052],[0,0,0,0],[8.999999E+09,8.999999E+09,8.999999E+09,8.999999E+09,8.999999E+09,8.999999E+09]];
	LOCAL CONST Robtarget Tr_meulage_motif_1_P299 :=[[35.737078125,-163.61415625,1.89253479003906],[0.696320279376617,-0.571579290814731,-0.275420255163045,0.335527742350052],[0,0,0,0],[8.999999E+09,8.999999E+09,8.999999E+09,8.999999E+09,8.999999E+09,8.999999E+09]];
	LOCAL CONST Robtarget Tr_meulage_motif_1_P300 :=[[36.333328125,-162.811359375,1.89255505371094],[0.696320279376617,-0.571579290814731,-0.275420255163045,0.335527742350052],[0,0,0,0],[8.999999E+09,8.999999E+09,8.999999E+09,8.999999E+09,8.999999E+09,8.999999E+09]];
	LOCAL CONST Robtarget Tr_meulage_motif_1_P301 :=[[36.929578125,-162.0085625,1.89257531738281],[0.696320279376617,-0.571579290814731,-0.275420255163045,0.335527742350052],[0,0,0,0],[8.999999E+09,8.999999E+09,8.999999E+09,8.999999E+09,8.999999E+09,8.999999E+09]];
	LOCAL CONST Robtarget Tr_meulage_motif_1_P302 :=[[37.5255234375,-161.214796875,1.78210559082031],[0.696320279376617,-0.571579290814731,-0.275420255163045,0.335527742350052],[0,0,0,0],[8.999999E+09,8.999999E+09,8.999999E+09,8.999999E+09,8.999999E+09,8.999999E+09]];
	LOCAL CONST Robtarget Tr_meulage_motif_1_P303 :=[[38.0977578125,-160.460796875,1.57116552734375],[0.696320279376617,-0.571579290814731,-0.275420255163045,0.335527742350052],[0,0,0,0],[8.999999E+09,8.999999E+09,8.999999E+09,8.999999E+09,8.999999E+09,8.999999E+09]];
	LOCAL CONST Robtarget Tr_meulage_motif_1_P304 :=[[38.6163359375,-159.783765625,1.2996484375],[0.696320279376617,-0.571579290814731,-0.275420255163045,0.335527742350052],[0,0,0,0],[8.999999E+09,8.999999E+09,8.999999E+09,8.999999E+09,8.999999E+09,8.999999E+09]];
	LOCAL CONST Robtarget Tr_meulage_motif_1_P305 :=[[39.0737890625,-159.189359375,1.0240244140625],[0.696320279376617,-0.571579290814731,-0.275420255163045,0.335527742350052],[0,0,0,0],[8.999999E+09,8.999999E+09,8.999999E+09,8.999999E+09,8.999999E+09,8.999999E+09]];
	LOCAL CONST Robtarget Tr_meulage_motif_1_P306 :=[[39.75329296875,-158.3225,0.408587615966797],[0.696320279376617,-0.571579290814731,-0.275420255163045,0.335527742350052],[0,0,0,0],[8.999999E+09,8.999999E+09,8.999999E+09,8.999999E+09,8.999999E+09,8.999999E+09]];
	LOCAL CONST Robtarget Tr_meulage_motif_1_P307 :=[[40.39541796875,-157.524,-0.438116119384766],[0.696320279376617,-0.571579290814731,-0.275420255163045,0.335527742350052],[0,0,0,0],[8.999999E+09,8.999999E+09,8.999999E+09,8.999999E+09,8.999999E+09,8.999999E+09]];
	LOCAL CONST Robtarget Tr_meulage_motif_1_P308 :=[[40.93905078125,-156.871875,-1.46085168457031],[0.696320279376617,-0.571579290814731,-0.275420255163045,0.335527742350052],[0,0,0,0],[8.999999E+09,8.999999E+09,8.999999E+09,8.999999E+09,8.999999E+09,8.999999E+09]];
	LOCAL CONST Robtarget Tr_meulage_motif_1_P309 :=[[41.27178125,-156.510890625,-2.57586987304688],[0.696320279376617,-0.571579290814731,-0.275420255163045,0.335527742350052],[0,0,0,0],[8.999999E+09,8.999999E+09,8.999999E+09,8.999999E+09,8.999999E+09,8.999999E+09]];
	LOCAL CONST Robtarget Tr_meulage_motif_1_P310 :=[[41.31389453125,-156.5084375,-3.27105444335937],[0.696320279376617,-0.571579290814731,-0.275420255163045,0.335527742350052],[0,0,0,0],[8.999999E+09,8.999999E+09,8.999999E+09,8.999999E+09,8.999999E+09,8.999999E+09]];
	LOCAL CONST Robtarget Tr_meulage_motif_1_P311 :=[[41.338578125,-156.526765625,-3.93162109375],[0.696320279376617,-0.571579290814731,-0.275420255163045,0.335527742350052],[0,0,0,0],[8.999999E+09,8.999999E+09,8.999999E+09,8.999999E+09,8.999999E+09,8.999999E+09]];
	LOCAL CONST Robtarget Tr_meulage_motif_1_P312 :=[[41.33053515625,-156.589125,-4.59198583984375],[0.696320279376617,-0.571579290814731,-0.275420255163045,0.335527742350052],[0,0,0,0],[8.999999E+09,8.999999E+09,8.999999E+09,8.999999E+09,8.999999E+09,8.999999E+09]];
	LOCAL CONST Robtarget Tr_meulage_motif_1_P313 :=[[41.07459375,-157.019609375,-5.69253955078125],[0.696320279376617,-0.571579290814731,-0.275420255163045,0.335527742350052],[0,0,0,0],[8.999999E+09,8.999999E+09,8.999999E+09,8.999999E+09,8.999999E+09,8.999999E+09]];
	LOCAL CONST Robtarget Tr_meulage_motif_1_P314 :=[[40.60140625,-157.7351875,-6.698109375],[0.696320279376617,-0.571579290814731,-0.275420255163045,0.335527742350052],[0,0,0,0],[8.999999E+09,8.999999E+09,8.999999E+09,8.999999E+09,8.999999E+09,8.999999E+09]];
	LOCAL CONST Robtarget Tr_meulage_motif_1_P315 :=[[40.022140625,-158.579734375,-7.52609375],[0.696320279376617,-0.571579290814731,-0.275420255163045,0.335527742350052],[0,0,0,0],[8.999999E+09,8.999999E+09,8.999999E+09,8.999999E+09,8.999999E+09,8.999999E+09]];
	LOCAL CONST Robtarget Tr_meulage_motif_1_P316 :=[[39.627234375,-159.142296875,-7.9214453125],[0.696320279376617,-0.571579290814731,-0.275420255163045,0.335527742350052],[0,0,0,0],[8.999999E+09,8.999999E+09,8.999999E+09,8.999999E+09,8.999999E+09,8.999999E+09]];
	LOCAL CONST Robtarget Tr_meulage_motif_1_P317 :=[[38.95487890625,-160.0855625,-8.4084736328125],[0.696320279376617,-0.571579290814731,-0.275420255163045,0.335527742350052],[0,0,0,0],[8.999999E+09,8.999999E+09,8.999999E+09,8.999999E+09,8.999999E+09,8.999999E+09]];
	LOCAL CONST Robtarget Tr_meulage_motif_1_P318 :=[[38.46088671875,-160.771265625,-8.672314453125],[0.696320279376617,-0.571579290814731,-0.275420255163045,0.335527742350052],[0,0,0,0],[8.999999E+09,8.999999E+09,8.999999E+09,8.999999E+09,8.999999E+09,8.999999E+09]];
	LOCAL CONST Robtarget Tr_meulage_motif_1_P319 :=[[37.91281640625,-161.525140625,-8.8765966796875],[0.696320279376617,-0.571579290814731,-0.275420255163045,0.335527742350052],[0,0,0,0],[8.999999E+09,8.999999E+09,8.999999E+09,8.999999E+09,8.999999E+09,8.999999E+09]];
	LOCAL CONST Robtarget Tr_meulage_motif_1_P320 :=[[37.331609375,-162.316140625,-8.9850458984375],[0.696320279376617,-0.571579290814731,-0.275420255163045,0.335527742350052],[0,0,0,0],[8.999999E+09,8.999999E+09,8.999999E+09,8.999999E+09,8.999999E+09,8.999999E+09]];
	LOCAL CONST Robtarget Tr_meulage_motif_1_P321 :=[[36.743921875,-163.11603125,-9.0955556640625],[0.696320279376617,-0.571579290814731,-0.275420255163045,0.335527742350052],[0,0,0,0],[8.999999E+09,8.999999E+09,8.999999E+09,8.999999E+09,8.999999E+09,8.999999E+09]];
	LOCAL CONST Robtarget Tr_meulage_motif_1_P322 :=[[36.147671875,-163.91884375,-9.095576171875],[0.696320279376617,-0.571579290814731,-0.275420255163045,0.335527742350052],[0,0,0,0],[8.999999E+09,8.999999E+09,8.999999E+09,8.999999E+09,8.999999E+09,8.999999E+09]];
	LOCAL CONST Robtarget Tr_meulage_motif_1_P323 :=[[35.551421875,-164.721640625,-9.0955966796875],[0.696320279376617,-0.571579290814731,-0.275420255163045,0.335527742350052],[0,0,0,0],[8.999999E+09,8.999999E+09,8.999999E+09,8.999999E+09,8.999999E+09,8.999999E+09]];
	LOCAL CONST Robtarget Tr_meulage_motif_1_P324 :=[[34.955171875,-165.5244375,-9.0956171875],[0.696320279376617,-0.571579290814731,-0.275420255163045,0.335527742350052],[0,0,0,0],[8.999999E+09,8.999999E+09,8.999999E+09,8.999999E+09,8.999999E+09,8.999999E+09]];
	LOCAL CONST Robtarget Tr_meulage_motif_1_P325 :=[[34.358921875,-166.327234375,-9.09563671875],[0.696320279376617,-0.571579290814731,-0.275420255163045,0.335527742350052],[0,0,0,0],[8.999999E+09,8.999999E+09,8.999999E+09,8.999999E+09,8.999999E+09,8.999999E+09]];
	LOCAL CONST Robtarget Tr_meulage_motif_1_P326 :=[[33.762671875,-167.13003125,-9.0956572265625],[0.696320279376617,-0.571579290814731,-0.275420255163045,0.335527742350052],[0,0,0,0],[8.999999E+09,8.999999E+09,8.999999E+09,8.999999E+09,8.999999E+09,8.999999E+09]];
	LOCAL CONST Robtarget Tr_meulage_motif_1_P327 :=[[33.166421875,-167.932828125,-9.095677734375],[0.696320279376617,-0.571579290814731,-0.275420255163045,0.335527742350052],[0,0,0,0],[8.999999E+09,8.999999E+09,8.999999E+09,8.999999E+09,8.999999E+09,8.999999E+09]];
	LOCAL CONST Robtarget Tr_meulage_motif_1_P328 :=[[32.570171875,-168.735625,-9.0956982421875],[0.696320279376617,-0.571579290814731,-0.275420255163045,0.335527742350052],[0,0,0,0],[8.999999E+09,8.999999E+09,8.999999E+09,8.999999E+09,8.999999E+09,8.999999E+09]];
	LOCAL CONST Robtarget Tr_meulage_motif_1_P329 :=[[31.973919921875,-169.538421875,-9.0957177734375],[0.696320279376617,-0.571579290814731,-0.275420255163045,0.335527742350052],[0,0,0,0],[8.999999E+09,8.999999E+09,8.999999E+09,8.999999E+09,8.999999E+09,8.999999E+09]];
	LOCAL CONST Robtarget Tr_meulage_motif_1_P330 :=[[31.377669921875,-170.34121875,-9.09573828125],[0.696320279376617,-0.571579290814731,-0.275420255163045,0.335527742350052],[0,0,0,0],[8.999999E+09,8.999999E+09,8.999999E+09,8.999999E+09,8.999999E+09,8.999999E+09]];
	LOCAL CONST Robtarget Tr_meulage_motif_1_P331 :=[[30.781419921875,-171.144015625,-9.0957587890625],[0.696320279376617,-0.571579290814731,-0.275420255163045,0.335527742350052],[0,0,0,0],[8.999999E+09,8.999999E+09,8.999999E+09,8.999999E+09,8.999999E+09,8.999999E+09]];
	LOCAL CONST Robtarget Tr_meulage_motif_1_P332 :=[[30.185169921875,-171.946828125,-9.095779296875],[0.696320279376617,-0.571579290814731,-0.275420255163045,0.335527742350052],[0,0,0,0],[8.999999E+09,8.999999E+09,8.999999E+09,8.999999E+09,8.999999E+09,8.999999E+09]];
	LOCAL CONST Robtarget Tr_meulage_motif_1_P333 :=[[29.588919921875,-172.749625,-9.095798828125],[0.696320279376617,-0.571579290814731,-0.275420255163045,0.335527742350052],[0,0,0,0],[8.999999E+09,8.999999E+09,8.999999E+09,8.999999E+09,8.999999E+09,8.999999E+09]];
	LOCAL CONST Robtarget Tr_meulage_motif_1_P334 :=[[28.992669921875,-173.552421875,-9.0958193359375],[0.696320279376617,-0.571579290814731,-0.275420255163045,0.335527742350052],[0,0,0,0],[8.999999E+09,8.999999E+09,8.999999E+09,8.999999E+09,8.999999E+09,8.999999E+09]];
	LOCAL CONST Robtarget Tr_meulage_motif_1_P335 :=[[28.396419921875,-174.35521875,-9.09583984375],[0.696320279376617,-0.571579290814731,-0.275420255163045,0.335527742350052],[0,0,0,0],[8.999999E+09,8.999999E+09,8.999999E+09,8.999999E+09,8.999999E+09,8.999999E+09]];
	LOCAL CONST Robtarget Tr_meulage_motif_1_P336 :=[[27.80016796875,-175.158015625,-9.0958603515625],[0.696320279376617,-0.571579290814731,-0.275420255163045,0.335527742350052],[0,0,0,0],[8.999999E+09,8.999999E+09,8.999999E+09,8.999999E+09,8.999999E+09,8.999999E+09]];
	LOCAL CONST Robtarget Tr_meulage_motif_1_P337 :=[[27.20391796875,-175.9608125,-9.0958798828125],[0.696320279376617,-0.571579290814731,-0.275420255163045,0.335527742350052],[0,0,0,0],[8.999999E+09,8.999999E+09,8.999999E+09,8.999999E+09,8.999999E+09,8.999999E+09]];
	LOCAL CONST Robtarget Tr_meulage_motif_1_P338 :=[[26.60766796875,-176.763609375,-9.095900390625],[0.696320279376617,-0.571579290814731,-0.275420255163045,0.335527742350052],[0,0,0,0],[8.999999E+09,8.999999E+09,8.999999E+09,8.999999E+09,8.999999E+09,8.999999E+09]];
	LOCAL CONST Robtarget Tr_meulage_motif_1_P339 :=[[26.01141796875,-177.56640625,-9.0959208984375],[0.696320279376617,-0.571579290814731,-0.275420255163045,0.335527742350052],[0,0,0,0],[8.999999E+09,8.999999E+09,8.999999E+09,8.999999E+09,8.999999E+09,8.999999E+09]];
	LOCAL CONST Robtarget Tr_meulage_motif_1_P340 :=[[25.41516796875,-178.369203125,-9.09594140625],[0.696320279376617,-0.571579290814731,-0.275420255163045,0.335527742350052],[0,0,0,0],[8.999999E+09,8.999999E+09,8.999999E+09,8.999999E+09,8.999999E+09,8.999999E+09]];
	LOCAL CONST Robtarget Tr_meulage_motif_1_P341 :=[[24.81891796875,-179.172015625,-9.0959609375],[0.696320279376617,-0.571579290814731,-0.275420255163045,0.335527742350052],[0,0,0,0],[8.999999E+09,8.999999E+09,8.999999E+09,8.999999E+09,8.999999E+09,8.999999E+09]];
	LOCAL CONST Robtarget Tr_meulage_motif_1_P342 :=[[24.222666015625,-179.9748125,-9.0959814453125],[0.696320279376617,-0.571579290814731,-0.275420255163045,0.335527742350052],[0,0,0,0],[8.999999E+09,8.999999E+09,8.999999E+09,8.999999E+09,8.999999E+09,8.999999E+09]];
	LOCAL CONST Robtarget Tr_meulage_motif_1_P343 :=[[23.626416015625,-180.777609375,-9.096001953125],[0.696320279376617,-0.571579290814731,-0.275420255163045,0.335527742350052],[0,0,0,0],[8.999999E+09,8.999999E+09,8.999999E+09,8.999999E+09,8.999999E+09,8.999999E+09]];
	LOCAL CONST Robtarget Tr_meulage_motif_1_P344 :=[[23.030166015625,-181.58040625,-9.0960224609375],[0.696320279376617,-0.571579290814731,-0.275420255163045,0.335527742350052],[0,0,0,0],[8.999999E+09,8.999999E+09,8.999999E+09,8.999999E+09,8.999999E+09,8.999999E+09]];
	LOCAL CONST Robtarget Tr_meulage_motif_1_P345 :=[[22.433916015625,-182.383203125,-9.0960419921875],[0.696320279376617,-0.571579290814731,-0.275420255163045,0.335527742350052],[0,0,0,0],[8.999999E+09,8.999999E+09,8.999999E+09,8.999999E+09,8.999999E+09,8.999999E+09]];
	LOCAL CONST Robtarget Tr_meulage_motif_1_P346 :=[[21.837666015625,-183.186,-9.0960625],[0.696320279376617,-0.571579290814731,-0.275420255163045,0.335527742350052],[0,0,0,0],[8.999999E+09,8.999999E+09,8.999999E+09,8.999999E+09,8.999999E+09,8.999999E+09]];
	LOCAL CONST Robtarget Tr_meulage_motif_1_P347 :=[[21.241416015625,-183.988796875,-9.0960830078125],[0.696320279376617,-0.571579290814731,-0.275420255163045,0.335527742350052],[0,0,0,0],[8.999999E+09,8.999999E+09,8.999999E+09,8.999999E+09,8.999999E+09,8.999999E+09]];
	LOCAL CONST Robtarget Tr_meulage_motif_1_P348 :=[[20.645166015625,-184.79159375,-9.096103515625],[0.696320279376617,-0.571579290814731,-0.275420255163045,0.335527742350052],[0,0,0,0],[8.999999E+09,8.999999E+09,8.999999E+09,8.999999E+09,8.999999E+09,8.999999E+09]];
	LOCAL CONST Robtarget Tr_meulage_motif_1_P349 :=[[20.0489140625,-185.594390625,-9.096123046875],[0.696320279376617,-0.571579290814731,-0.275420255163045,0.335527742350052],[0,0,0,0],[8.999999E+09,8.999999E+09,8.999999E+09,8.999999E+09,8.999999E+09,8.999999E+09]];
	LOCAL CONST Robtarget Tr_meulage_motif_1_P350 :=[[19.4526640625,-186.397203125,-9.0961435546875],[0.696320279376617,-0.571579290814731,-0.275420255163045,0.335527742350052],[0,0,0,0],[8.999999E+09,8.999999E+09,8.999999E+09,8.999999E+09,8.999999E+09,8.999999E+09]];
	LOCAL CONST Robtarget Tr_meulage_motif_1_P351 :=[[18.8564140625,-187.2,-9.0961640625],[0.696320279376617,-0.571579290814731,-0.275420255163045,0.335527742350052],[0,0,0,0],[8.999999E+09,8.999999E+09,8.999999E+09,8.999999E+09,8.999999E+09,8.999999E+09]];
	LOCAL CONST Robtarget Tr_meulage_motif_1_P352 :=[[18.2601640625,-188.002796875,-9.0961845703125],[0.696320279376617,-0.571579290814731,-0.275420255163045,0.335527742350052],[0,0,0,0],[8.999999E+09,8.999999E+09,8.999999E+09,8.999999E+09,8.999999E+09,8.999999E+09]];
	LOCAL CONST Robtarget Tr_meulage_motif_1_P353 :=[[17.6639140625,-188.80559375,-9.0962041015625],[0.696320279376617,-0.571579290814731,-0.275420255163045,0.335527742350052],[0,0,0,0],[8.999999E+09,8.999999E+09,8.999999E+09,8.999999E+09,8.999999E+09,8.999999E+09]];
	LOCAL CONST Robtarget Tr_meulage_motif_1_P354 :=[[17.0676640625,-189.608390625,-9.096224609375],[0.696320279376617,-0.571579290814731,-0.275420255163045,0.335527742350052],[0,0,0,0],[8.999999E+09,8.999999E+09,8.999999E+09,8.999999E+09,8.999999E+09,8.999999E+09]];
	LOCAL CONST Robtarget Tr_meulage_motif_1_P355 :=[[16.4714140625,-190.4111875,-9.0962451171875],[0.696320279376617,-0.571579290814731,-0.275420255163045,0.335527742350052],[0,0,0,0],[8.999999E+09,8.999999E+09,8.999999E+09,8.999999E+09,8.999999E+09,8.999999E+09]];
	LOCAL CONST Robtarget Tr_meulage_motif_1_P356 :=[[15.8751630859375,-191.213984375,-9.096265625],[0.696320279376617,-0.571579290814731,-0.275420255163045,0.335527742350052],[0,0,0,0],[8.999999E+09,8.999999E+09,8.999999E+09,8.999999E+09,8.999999E+09,8.999999E+09]];
	LOCAL CONST Robtarget Tr_meulage_motif_1_P357 :=[[15.278912109375,-192.01678125,-9.09628515625],[0.696320279376617,-0.571579290814731,-0.275420255163045,0.335527742350052],[0,0,0,0],[8.999999E+09,8.999999E+09,8.999999E+09,8.999999E+09,8.999999E+09,8.999999E+09]];
	LOCAL CONST Robtarget Tr_meulage_motif_1_P358 :=[[14.682662109375,-192.819578125,-9.0963056640625],[0.696320279376617,-0.571579290814731,-0.275420255163045,0.335527742350052],[0,0,0,0],[8.999999E+09,8.999999E+09,8.999999E+09,8.999999E+09,8.999999E+09,8.999999E+09]];
	LOCAL CONST Robtarget Tr_meulage_motif_1_P359 :=[[14.086412109375,-193.622390625,-9.096326171875],[0.696320279376617,-0.571579290814731,-0.275420255163045,0.335527742350052],[0,0,0,0],[8.999999E+09,8.999999E+09,8.999999E+09,8.999999E+09,8.999999E+09,8.999999E+09]];
	LOCAL CONST Robtarget Tr_meulage_motif_1_P360 :=[[13.490162109375,-194.4251875,-9.0963466796875],[0.696320279376617,-0.571579290814731,-0.275420255163045,0.335527742350052],[0,0,0,0],[8.999999E+09,8.999999E+09,8.999999E+09,8.999999E+09,8.999999E+09,8.999999E+09]];
	LOCAL CONST Robtarget Tr_meulage_motif_1_P361 :=[[12.8939111328125,-195.227984375,-9.0963662109375],[0.696320279376617,-0.571579290814731,-0.275420255163045,0.335527742350052],[0,0,0,0],[8.999999E+09,8.999999E+09,8.999999E+09,8.999999E+09,8.999999E+09,8.999999E+09]];
	LOCAL CONST Robtarget Tr_meulage_motif_1_P362 :=[[12.2976611328125,-196.03078125,-9.09638671875],[0.696320279376617,-0.571579290814731,-0.275420255163045,0.335527742350052],[0,0,0,0],[8.999999E+09,8.999999E+09,8.999999E+09,8.999999E+09,8.999999E+09,8.999999E+09]];
	LOCAL CONST Robtarget Tr_meulage_motif_1_P363 :=[[11.7014111328125,-196.833578125,-9.0964072265625],[0.696320279376617,-0.571579290814731,-0.275420255163045,0.335527742350052],[0,0,0,0],[8.999999E+09,8.999999E+09,8.999999E+09,8.999999E+09,8.999999E+09,8.999999E+09]];
	LOCAL CONST Robtarget Tr_meulage_motif_1_P364 :=[[11.10516015625,-197.636375,-9.096427734375],[0.696320279376617,-0.571579290814731,-0.275420255163045,0.335527742350052],[0,0,0,0],[8.999999E+09,8.999999E+09,8.999999E+09,8.999999E+09,8.999999E+09,8.999999E+09]];
	LOCAL CONST Robtarget Tr_meulage_motif_1_P365 :=[[10.5174736328125,-198.436265625,-9.2069375],[0.696320279376617,-0.571579290814731,-0.275420255163045,0.335527742350052],[0,0,0,0],[8.999999E+09,8.999999E+09,8.999999E+09,8.999999E+09,8.999999E+09,8.999999E+09]];
	LOCAL CONST Robtarget Tr_meulage_motif_1_P366 :=[[9.961005859375,-199.20196875,-9.417916015625],[0.696320279376617,-0.571579290814731,-0.275420255163045,0.335527742350052],[0,0,0,0],[8.999999E+09,8.999999E+09,8.999999E+09,8.999999E+09,8.999999E+09,8.999999E+09]];
	LOCAL CONST Robtarget Tr_meulage_motif_1_P367 :=[[9.4627177734375,-199.8940625,-9.6894677734375],[0.696320279376617,-0.571579290814731,-0.275420255163045,0.335527742350052],[0,0,0,0],[8.999999E+09,8.999999E+09,8.999999E+09,8.999999E+09,8.999999E+09,8.999999E+09]];
	LOCAL CONST Robtarget Tr_meulage_motif_1_P368 :=[[9.0498388671875,-200.473671875,-9.9932939453125],[0.696320279376617,-0.571579290814731,-0.275420255163045,0.335527742350052],[0,0,0,0],[8.999999E+09,8.999999E+09,8.999999E+09,8.999999E+09,8.999999E+09,8.999999E+09]];
	LOCAL CONST Robtarget Tr_meulage_motif_1_P369 :=[[8.4577666015625,-201.3225,-10.6551298828125],[0.696320279376617,-0.571579290814731,-0.275420255163045,0.335527742350052],[0,0,0,0],[8.999999E+09,8.999999E+09,8.999999E+09,8.999999E+09,8.999999E+09,8.999999E+09]];
	LOCAL CONST Robtarget Tr_meulage_motif_1_P370 :=[[8.0081689453125,-202.00109375,-11.593912109375],[0.696320279376617,-0.571579290814731,-0.275420255163045,0.335527742350052],[0,0,0,0],[8.999999E+09,8.999999E+09,8.999999E+09,8.999999E+09,8.999999E+09,8.999999E+09]];
	LOCAL CONST Robtarget Tr_meulage_motif_1_P371 :=[[7.83521875,-202.311625,-12.589201171875],[0.696320279376617,-0.571579290814731,-0.275420255163045,0.335527742350052],[0,0,0,0],[8.999999E+09,8.999999E+09,8.999999E+09,8.999999E+09,8.999999E+09,8.999999E+09]];
	LOCAL CONST Robtarget Tr_meulage_motif_1_P372 :=[[7.8737314453125,-202.303234375,-13.1461455078125],[0.696320279376617,-0.571579290814731,-0.275420255163045,0.335527742350052],[0,0,0,0],[8.999999E+09,8.999999E+09,8.999999E+09,8.999999E+09,8.999999E+09,8.999999E+09]];
	LOCAL CONST Robtarget Tr_meulage_motif_1_P373 :=[[7.886740234375,-202.318296875,-13.563599609375],[0.696320279376617,-0.571579290814731,-0.275420255163045,0.335527742350052],[0,0,0,0],[8.999999E+09,8.999999E+09,8.999999E+09,8.999999E+09,8.999999E+09,8.999999E+09]];
